KUKA KRL program: EPS_2_251349_CBMH080_A_20251001124254.src

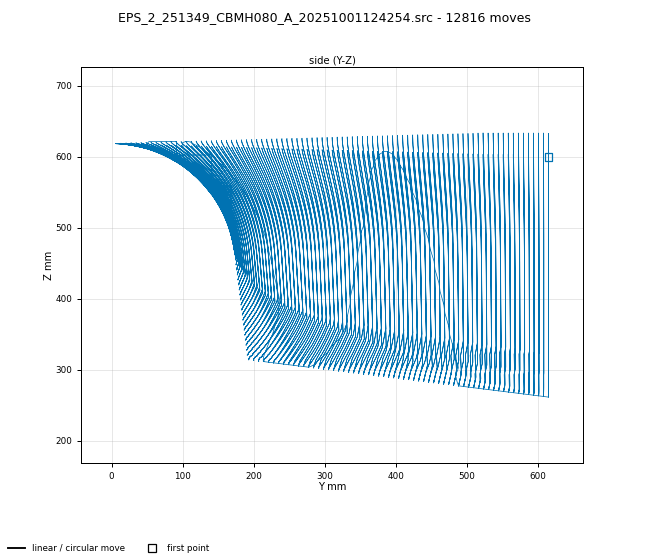
[picture p0: tool path of EPS_2_251349_CBMH080_A_20251001124254.src, 12816 of 12818 moves have a stored position in this frame; points joined in program order, loops and branches not executed]
&ACCESS RVP
&REL 4
&COMMENT QRS 19112012
&PARAM EDITMASK = *
DEF PART()
EXT BAS (BAS_COMMAND :IN,REAL :IN )
INT I
BAS (#INITMOV,0 )

;KUKA QRS Post kuka4.cps  Date:22-06-2017 !

File_ID=2857

QRS_PRE_INIT()

;Init var - Until changes are made in qrs_pre_init
Outlet_Square_prg=0
Inlet_1_Square_prg=0
Inlet_2_Square_prg=0
Inlet_3_Square_prg=0
Inlet_4_Square_prg=0
Inlet_5_Square_prg=0

Outlet_1={X 0.000, Y 523.550, Z 484.000, B 0.000, E1 0.000 }
Inlet_1={X 0.000, Y 525.740, Z 454.000, B 0.000, E1 180.000 }
Outlet_1_type=299
Inlet_1_type=299
;QRS#1=Sidecore dimensions
;QRS#2=300-12" PVC SDR 35
;QRS#3=300-12" PVC SDR 35
;QRS#4=
;QRS#5=
;QRS#6=
;QRS#7=
;QRS#8=
;QRS#9=16M PSX
;QRS#10=16M PSX
;QRS#11=
;QRS#12=
;QRS#13=
;QRS#14=
;QRS#15=
;QRS#16=1220x127x914 3'
;QRS#17=EPS Height
;QRS#18=633,5
;QRS#19=*
;QRS#20= UPDATED VERSION 22-06-2017
;QRS#21=*
Outlet_Square=0150
Inlet_1_Square=0150
Inlet_2_Square=0
Inlet_3_Square=0
Inlet_4_Square=0
Inlet_5_Square=0
Mill_Square=1
Outlet_Square_Prg=206
Inlet_1_Square_prg=206

QRS_INIT()

$ADVANCE=5

; T1
PTP {E1 173.644,E2 173.644}
PTP {X 0,Y 615.424,A -85,B 0,C 180,E1 173.644,E2 173.644,E3 0,E4 0,E5 0,E6 0}
QRS_SPEED_INIT()
LIN {X 0,Y 615.424,Z 600,A -85,B 0,C 180,E1 173.644,E2 173.644,E3 0,E4 0,E5 0,E6 0} C_VEL
LIN {X 0,Y 615.424,Z 271.5,A -85,B 0,C 180,E1 173.644,E2 173.644} C_VEL
LIN {X 0,Y 615.424,Z 263.323,A -85,B 0,C 180,E1 173.644,E2 173.644} C_VEL
LIN {X 0,Y 615.426,Z 261.323,A -85,B 0,C 180,E1 173.458,E2 173.458} C_VEL
LIN {X 0,Y 615.491,Z 261.325,A -85,B 0,C 180,E1 170.801,E2 170.801} C_VEL
LIN {X 0,Y 615.447,Z 261.319,A -85,B 0,C 180,E1 168.138,E2 168.138} C_VEL
LIN {X 0,Y 615.442,Z 261.319,A -85,B 0,C 180,E1 166.078,E2 166.078} C_VEL
LIN {X 0,Y 615.442,Z 261.319,A -85,B 0,C 180,E1 164.094,E2 164.094} C_VEL
LIN {X 0,Y 615.44,Z 261.319,A -85,B 0,C 180,E1 162.042,E2 162.042} C_VEL
LIN {X 0,Y 615.435,Z 261.319,A -85,B 0,C 180,E1 159.965,E2 159.965} C_VEL
LIN {X 0,Y 615.434,Z 261.321,A -85,B 0,C 180,E1 157.662,E2 157.662} C_VEL
LIN {X 0,Y 615.491,Z 261.325,A -85,B 0,C 180,E1 155.008,E2 155.008} C_VEL
LIN {X 0,Y 615.494,Z 261.32,A -85,B 0,C 180,E1 152.823,E2 152.823} C_VEL
LIN {X 0,Y 615.451,Z 261.316,A -85,B 0,C 180,E1 150.209,E2 150.209} C_VEL
LIN {X 0,Y 615.44,Z 261.321,A -85,B 0,C 180,E1 147.674,E2 147.674} C_VEL
LIN {X 0,Y 615.485,Z 261.325,A -85,B 0,C 180,E1 145.185,E2 145.185} C_VEL
LIN {X 0,Y 615.491,Z 261.315,A -85,B 0,C 180,E1 142.758,E2 142.758} C_VEL
LIN {X 0,Y 615.453,Z 261.315,A -85,B 0,C 180,E1 140.247,E2 140.247} C_VEL
LIN {X 0,Y 615.455,Z 261.321,A -85,B 0,C 180,E1 137.644,E2 137.644} C_VEL
LIN {X 0,Y 615.489,Z 261.317,A -85,B 0,C 180,E1 134.931,E2 134.931} C_VEL
LIN {X 0,Y 615.455,Z 261.315,A -85,B 0,C 180,E1 132.354,E2 132.354} C_VEL
LIN {X 0,Y 615.457,Z 261.32,A -85,B 0,C 180,E1 129.751,E2 129.751} C_VEL
LIN {X 0,Y 615.488,Z 261.315,A -85,B 0,C 180,E1 126.937,E2 126.937} C_VEL
LIN {X 0,Y 615.453,Z 261.318,A -85,B 0,C 180,E1 124.023,E2 124.023} C_VEL
LIN {X 0,Y 615.492,Z 261.316,A -85,B 0,C 180,E1 121.086,E2 121.086} C_VEL
LIN {X 0,Y 615.462,Z 261.313,A -85,B 0,C 180,E1 118.446,E2 118.446} C_VEL
LIN {X 0,Y 615.476,Z 261.322,A -85,B 0,C 180,E1 115.715,E2 115.715} C_VEL
LIN {X 0,Y 615.486,Z 261.31,A -85,B 0,C 180,E1 112.844,E2 112.844} C_VEL
LIN {X 0,Y 615.459,Z 261.362,A -85,B 0,C 180,E1 112.263,E2 112.263} C_VEL
LIN {X 0,Y 615.464,Z 281.213,A -85,B 0,C 180,E1 109.685,E2 109.685} C_VEL
LIN {X 0,Y 615.457,Z 292.799,A -85,B 0,C 180,E1 108.199,E2 108.199} C_VEL
LIN {X 0,Y 615.489,Z 457.351,A -85,B 0,C 180,E1 106.199,E2 106.199} C_VEL
LIN {X 0,Y 615.489,Z 471.838,A -85,B 0,C 180,E1 105.905,E2 105.905} C_VEL
LIN {X 0,Y 615.477,Z 486.432,A -85,B 0,C 180,E1 105.48,E2 105.48} C_VEL
LIN {X 0,Y 615.491,Z 499.749,A -85,B 0,C 180,E1 104.971,E2 104.971} C_VEL
LIN {X 0,Y 615.483,Z 513.386,A -85,B 0,C 180,E1 104.319,E2 104.319} C_VEL
LIN {X 0,Y 615.5,Z 526.673,A -85,B 0,C 180,E1 103.537,E2 103.537} C_VEL
LIN {X 0,Y 615.497,Z 538.522,A -85,B 0,C 180,E1 102.697,E2 102.697} C_VEL
LIN {X 0,Y 615.497,Z 550.364,A -85,B 0,C 180,E1 101.693,E2 101.693} C_VEL
LIN {X 0,Y 615.495,Z 560.168,A -85,B 0,C 180,E1 100.708,E2 100.708} C_VEL
LIN {X 0,Y 615.495,Z 570.015,A -85,B 0,C 180,E1 99.53,E2 99.53} C_VEL
LIN {X 0,Y 615.497,Z 578.104,A -85,B 0,C 180,E1 98.371,E2 98.371} C_VEL
LIN {X 0,Y 615.491,Z 584.784,A -85,B 0,C 180,E1 97.215,E2 97.215} C_VEL
LIN {X 0,Y 615.497,Z 590.949,A -85,B 0,C 180,E1 95.898,E2 95.898} C_VEL
LIN {X 0,Y 615.49,Z 595.717,A -85,B 0,C 180,E1 94.584,E2 94.584} C_VEL
LIN {X 0,Y 615.491,Z 599.221,A -85,B 0,C 180,E1 93.273,E2 93.273} C_VEL
LIN {X 0,Y 615.499,Z 601.54,A -85,B 0,C 180,E1 91.963,E2 91.963} C_VEL
LIN {X 0,Y 615.491,Z 602.728,A -85,B 0,C 180,E1 90.654,E2 90.654} C_VEL
LIN {X 0,Y 615.492,Z 602.751,A -85,B 0,C 180,E1 89.346,E2 89.346} C_VEL
LIN {X 0,Y 615.499,Z 601.646,A -85,B 0,C 180,E1 88.037,E2 88.037} C_VEL
LIN {X 0,Y 615.494,Z 599.416,A -85,B 0,C 180,E1 86.727,E2 86.727} C_VEL
LIN {X 0,Y 615.491,Z 596.005,A -85,B 0,C 180,E1 85.416,E2 85.416} C_VEL
LIN {X 0,Y 615.498,Z 591.336,A -85,B 0,C 180,E1 84.102,E2 84.102} C_VEL
LIN {X 0,Y 615.49,Z 585.273,A -85,B 0,C 180,E1 82.785,E2 82.785} C_VEL
LIN {X 0,Y 615.49,Z 577.635,A -85,B 0,C 180,E1 81.464,E2 81.464} C_VEL
LIN {X 0,Y 615.495,Z 569.452,A -85,B 0,C 180,E1 80.304,E2 80.304} C_VEL
LIN {X 0,Y 615.496,Z 559.333,A -85,B 0,C 180,E1 79.109,E2 79.109} C_VEL
LIN {X 0,Y 615.498,Z 547.686,A -85,B 0,C 180,E1 77.973,E2 77.973} C_VEL
LIN {X 0,Y 615.498,Z 536.417,A -85,B 0,C 180,E1 77.051,E2 77.051} C_VEL
LIN {X 0,Y 615.498,Z 524.179,A -85,B 0,C 180,E1 76.211,E2 76.211} C_VEL
LIN {X 0,Y 615.48,Z 510.782,A -85,B 0,C 180,E1 75.451,E2 75.451} C_VEL
LIN {X 0,Y 615.493,Z 496.919,A -85,B 0,C 180,E1 74.817,E2 74.817} C_VEL
LIN {X 0,Y 615.488,Z 482.706,A -85,B 0,C 180,E1 74.308,E2 74.308} C_VEL
LIN {X 0,Y 615.497,Z 468.664,A -85,B 0,C 180,E1 73.932,E2 73.932} C_VEL
LIN {X 0,Y 615.487,Z 453.239,A -85,B 0,C 180,E1 73.653,E2 73.653} C_VEL
LIN {X 0,Y 615.457,Z 292.88,A -85,B 0,C 180,E1 71.721,E2 71.721} C_VEL
LIN {X 0,Y 615.49,Z 271.117,A -85,B 0,C 180,E1 68.92,E2 68.92} C_VEL
LIN {X 0,Y 615.465,Z 261.314,A -85,B 0,C 180,E1 67.628,E2 67.628} C_VEL
LIN {X 0,Y 615.491,Z 261.31,A -85,B 0,C 180,E1 65.009,E2 65.009} C_VEL
LIN {X 0,Y 615.467,Z 261.32,A -85,B 0,C 180,E1 62.085,E2 62.085} C_VEL
LIN {X 0,Y 615.458,Z 261.316,A -85,B 0,C 180,E1 59.839,E2 59.839} C_VEL
LIN {X 0,Y 615.468,Z 261.312,A -85,B 0,C 180,E1 57.542,E2 57.542} C_VEL
LIN {X 0,Y 615.499,Z 261.308,A -85,B 0,C 180,E1 55.187,E2 55.187} C_VEL
LIN {X 0,Y 615.493,Z 261.321,A -85,B 0,C 180,E1 52.759,E2 52.759} C_VEL
LIN {X 0,Y 615.465,Z 261.321,A -85,B 0,C 180,E1 50.249,E2 50.249} C_VEL
LIN {X 0,Y 615.458,Z 261.314,A -85,B 0,C 180,E1 47.646,E2 47.646} C_VEL
LIN {X 0,Y 615.489,Z 261.319,A -85,B 0,C 180,E1 44.933,E2 44.933} C_VEL
LIN {X 0,Y 615.462,Z 261.321,A -85,B 0,C 180,E1 42.355,E2 42.355} C_VEL
LIN {X 0,Y 615.456,Z 261.315,A -85,B 0,C 180,E1 39.753,E2 39.753} C_VEL
LIN {X 0,Y 615.489,Z 261.323,A -85,B 0,C 180,E1 36.939,E2 36.939} C_VEL
LIN {X 0,Y 615.446,Z 261.317,A -85,B 0,C 180,E1 34.025,E2 34.025} C_VEL
LIN {X 0,Y 615.492,Z 261.32,A -85,B 0,C 180,E1 31.089,E2 31.089} C_VEL
LIN {X 0,Y 615.451,Z 261.321,A -85,B 0,C 180,E1 28.447,E2 28.447} C_VEL
LIN {X 0,Y 615.449,Z 261.321,A -85,B 0,C 180,E1 26.446,E2 26.446} C_VEL
LIN {X 0,Y 615.442,Z 261.318,A -85,B 0,C 180,E1 24.002,E2 24.002} C_VEL
LIN {X 0,Y 615.491,Z 261.314,A -85,B 0,C 180,E1 21.432,E2 21.432} C_VEL
LIN {X 0,Y 615.448,Z 261.322,A -85,B 0,C 180,E1 18.599,E2 18.599} C_VEL
LIN {X 0,Y 615.436,Z 261.321,A -85,B 0,C 180,E1 16.42,E2 16.42} C_VEL
LIN {X 0,Y 615.44,Z 261.322,A -85,B 0,C 180,E1 14.55,E2 14.55} C_VEL
LIN {X 0,Y 615.437,Z 261.322,A -85,B 0,C 180,E1 12.531,E2 12.531} C_VEL
LIN {X 0,Y 615.434,Z 261.322,A -85,B 0,C 180,E1 10.528,E2 10.528} C_VEL
LIN {X 0,Y 615.429,Z 261.323,A -85,B 0,C 180,E1 8.538,E2 8.538} C_VEL
LIN {X 0,Y 615.431,Z 261.322,A -85,B 0,C 180,E1 6.546,E2 6.546} C_VEL
LIN {X 0,Y 615.427,Z 261.323,A -85,B 0,C 180,E1 4.585,E2 4.585} C_VEL
LIN {X 0,Y 615.43,Z 261.323,A -85,B 0,C 180,E1 2.618,E2 2.618} C_VEL
LIN {X 0,Y 615.429,Z 261.323,A -85,B 0,C 180,E1 0.654,E2 0.654} C_VEL
LIN {X 0,Y 615.428,Z 261.323,A -85,B 0,C 180,E1 -1.309,E2 -1.309} C_VEL
LIN {X 0,Y 615.428,Z 261.323,A -85,B 0,C 180,E1 -3.273,E2 -3.273} C_VEL
LIN {X 0,Y 615.426,Z 261.324,A -85,B 0,C 180,E1 -5.242,E2 -5.242} C_VEL
LIN {X 0,Y 615.426,Z 261.324,A -85,B 0,C 180,E1 -7.216,E2 -7.216} C_VEL
LIN {X 0,Y 615.423,Z 261.324,A -85,B 0,C 180,E1 -9.2,E2 -9.2} C_VEL
LIN {X 0,Y 615.422,Z 261.324,A -85,B 0,C 180,E1 -11.194,E2 -11.194} C_VEL
LIN {X 0,Y 615.419,Z 261.324,A -85,B 0,C 180,E1 -13.203,E2 -13.203} C_VEL
LIN {X 0,Y 615.416,Z 261.325,A -85,B 0,C 180,E1 -15.228,E2 -15.228} C_VEL
LIN {X 0,Y 615.412,Z 261.325,A -85,B 0,C 180,E1 -17.273,E2 -17.273} C_VEL
LIN {X 0,Y 615.41,Z 261.325,A -85,B 0,C 180,E1 -19.34,E2 -19.34} C_VEL
LIN {X 0,Y 615.411,Z 261.325,A -85,B 0,C 180,E1 -21.435,E2 -21.435} C_VEL
LIN {X 0,Y 615.416,Z 261.325,A -85,B 0,C 180,E1 -23.559,E2 -23.559} C_VEL
LIN {X 0,Y 615.485,Z 261.323,A -85,B 0,C 180,E1 -26.444,E2 -26.444} C_VEL
LIN {X 0,Y 615.454,Z 261.322,A -85,B 0,C 180,E1 -28.66,E2 -28.66} C_VEL
LIN {X 0,Y 615.422,Z 261.323,A -85,B 0,C 180,E1 -31.078,E2 -31.078} C_VEL
LIN {X 0,Y 615.42,Z 261.323,A -85,B 0,C 180,E1 -33.24,E2 -33.24} C_VEL
LIN {X 0,Y 615.454,Z 261.324,A -85,B 0,C 180,E1 -35.832,E2 -35.832} C_VEL
LIN {X 0,Y 615.486,Z 261.326,A -85,B 0,C 180,E1 -38.069,E2 -38.069} C_VEL
LIN {X 0,Y 615.455,Z 261.32,A -85,B 0,C 180,E1 -40.609,E2 -40.609} C_VEL
LIN {X 0,Y 615.428,Z 261.321,A -85,B 0,C 180,E1 -43.043,E2 -43.043} C_VEL
LIN {X 0,Y 615.428,Z 261.321,A -85,B 0,C 180,E1 -45.074,E2 -45.074} C_VEL
LIN {X 0,Y 615.455,Z 261.323,A -85,B 0,C 180,E1 -47.646,E2 -47.646} C_VEL
LIN {X 0,Y 615.492,Z 261.317,A -85,B 0,C 180,E1 -50.252,E2 -50.252} C_VEL
LIN {X 0,Y 615.441,Z 261.318,A -85,B 0,C 180,E1 -52.756,E2 -52.756} C_VEL
LIN {X 0,Y 615.437,Z 261.321,A -85,B 0,C 180,E1 -55.183,E2 -55.183} C_VEL
LIN {X 0,Y 615.476,Z 261.324,A -85,B 0,C 180,E1 -57.671,E2 -57.671} C_VEL
LIN {X 0,Y 615.453,Z 261.316,A -85,B 0,C 180,E1 -60.593,E2 -60.593} C_VEL
LIN {X 0,Y 615.44,Z 261.319,A -85,B 0,C 180,E1 -62.964,E2 -62.964} C_VEL
LIN {X 0,Y 615.441,Z 261.446,A -85,B 0,C 180,E1 -64.936,E2 -64.936} C_VEL
LIN {X 0,Y 615.482,Z 284.083,A -85,B 0,C 180,E1 -67.53,E2 -67.53} C_VEL
LIN {X 0,Y 615.49,Z 308.881,A -85,B 0,C 180,E1 -70.316,E2 -70.316} C_VEL
LIN {X 0,Y 615.488,Z 322.06,A -85,B 0,C 180,E1 -71.762,E2 -71.762} C_VEL
LIN {X 0,Y 615.487,Z 488.129,A -85,B 0,C 180,E1 -73.767,E2 -73.767} C_VEL
LIN {X 0,Y 615.49,Z 503.731,A -85,B 0,C 180,E1 -74.095,E2 -74.095} C_VEL
LIN {X 0,Y 615.48,Z 519.063,A -85,B 0,C 180,E1 -74.562,E2 -74.562} C_VEL
LIN {X 0,Y 615.492,Z 532.764,A -85,B 0,C 180,E1 -75.113,E2 -75.113} C_VEL
LIN {X 0,Y 615.494,Z 547.049,A -85,B 0,C 180,E1 -75.834,E2 -75.834} C_VEL
LIN {X 0,Y 615.497,Z 559.904,A -85,B 0,C 180,E1 -76.631,E2 -76.631} C_VEL
LIN {X 0,Y 615.495,Z 572.259,A -85,B 0,C 180,E1 -77.554,E2 -77.554} C_VEL
LIN {X 0,Y 615.495,Z 582.61,A -85,B 0,C 180,E1 -78.474,E2 -78.474} C_VEL
LIN {X 0,Y 615.495,Z 592.187,A -85,B 0,C 180,E1 -79.474,E2 -79.474} C_VEL
LIN {X 0,Y 615.494,Z 601.579,A -85,B 0,C 180,E1 -80.636,E2 -80.636} C_VEL
LIN {X 0,Y 615.495,Z 609.382,A -85,B 0,C 180,E1 -81.794,E2 -81.794} C_VEL
LIN {X 0,Y 615.496,Z 616.607,A -85,B 0,C 180,E1 -83.102,E2 -83.102} C_VEL
LIN {X 0,Y 615.499,Z 622.437,A -85,B 0,C 180,E1 -84.43,E2 -84.43} C_VEL
LIN {X 0,Y 615.491,Z 625.861,A -85,B 0,C 180,E1 -85.416,E2 -85.416} C_VEL
LIN {X 0,Y 615.492,Z 629.318,A -85,B 0,C 180,E1 -86.727,E2 -86.727} C_VEL
LIN {X 0,Y 615.497,Z 631.593,A -85,B 0,C 180,E1 -88.037,E2 -88.037} C_VEL
LIN {X 0,Y 615.493,Z 632.74,A -85,B 0,C 180,E1 -89.346,E2 -89.346} C_VEL
LIN {X 0,Y 615.493,Z 632.74,A -85,B 0,C 180,E1 -90.654,E2 -90.654} C_VEL
LIN {X 0,Y 615.497,Z 631.593,A -85,B 0,C 180,E1 -91.963,E2 -91.963} C_VEL
LIN {X 0,Y 615.492,Z 629.318,A -85,B 0,C 180,E1 -93.273,E2 -93.273} C_VEL
LIN {X 0,Y 615.491,Z 625.861,A -85,B 0,C 180,E1 -94.584,E2 -94.584} C_VEL
LIN {X 0,Y 615.49,Z 621.144,A -85,B 0,C 180,E1 -95.898,E2 -95.898} C_VEL
LIN {X 0,Y 615.495,Z 615.03,A -85,B 0,C 180,E1 -97.215,E2 -97.215} C_VEL
LIN {X 0,Y 615.49,Z 607.335,A -85,B 0,C 180,E1 -98.536,E2 -98.536} C_VEL
LIN {X 0,Y 615.495,Z 599.116,A -85,B 0,C 180,E1 -99.696,E2 -99.696} C_VEL
LIN {X 0,Y 615.497,Z 588.895,A -85,B 0,C 180,E1 -100.893,E2 -100.893} C_VEL
LIN {X 0,Y 615.495,Z 579.071,A -85,B 0,C 180,E1 -101.86,E2 -101.86} C_VEL
LIN {X 0,Y 615.498,Z 566.952,A -85,B 0,C 180,E1 -102.865,E2 -102.865} C_VEL
LIN {X 0,Y 615.498,Z 554.804,A -85,B 0,C 180,E1 -103.705,E2 -103.705} C_VEL
LIN {X 0,Y 615.484,Z 541.386,A -85,B 0,C 180,E1 -104.472,E2 -104.472} C_VEL
LIN {X 0,Y 615.495,Z 526.858,A -85,B 0,C 180,E1 -105.141,E2 -105.141} C_VEL
LIN {X 0,Y 615.484,Z 512.629,A -85,B 0,C 180,E1 -105.65,E2 -105.65} C_VEL
LIN {X 0,Y 615.499,Z 498.141,A -85,B 0,C 180,E1 -106.035,E2 -106.035} C_VEL
LIN {X 0,Y 615.487,Z 483.539,A -85,B 0,C 180,E1 -106.298,E2 -106.298} C_VEL
LIN {X 0,Y 615.489,Z 321.746,A -85,B 0,C 180,E1 -108.258,E2 -108.258} C_VEL
LIN {X 0,Y 615.49,Z 296.397,A -85,B 0,C 180,E1 -111.08,E2 -111.08} C_VEL
LIN {X 0,Y 615.495,Z 270.579,A -85,B 0,C 180,E1 -114.01,E2 -114.01} C_VEL
LIN {X 0,Y 615.441,Z 261.318,A -85,B 0,C 180,E1 -115.1,E2 -115.1} C_VEL
LIN {X 0,Y 615.489,Z 261.317,A -85,B 0,C 180,E1 -117.914,E2 -117.914} C_VEL
LIN {X 0,Y 615.499,Z 261.324,A -85,B 0,C 180,E1 -120.159,E2 -120.159} C_VEL
LIN {X 0,Y 615.462,Z 261.323,A -85,B 0,C 180,E1 -122.458,E2 -122.458} C_VEL
LIN {X 0,Y 615.437,Z 261.321,A -85,B 0,C 180,E1 -124.817,E2 -124.817} C_VEL
LIN {X 0,Y 615.442,Z 261.318,A -85,B 0,C 180,E1 -127.244,E2 -127.244} C_VEL
LIN {X 0,Y 615.495,Z 261.325,A -85,B 0,C 180,E1 -130.09,E2 -130.09} C_VEL
LIN {X 0,Y 615.457,Z 261.323,A -85,B 0,C 180,E1 -132.354,E2 -132.354} C_VEL
LIN {X 0,Y 615.429,Z 261.321,A -85,B 0,C 180,E1 -134.926,E2 -134.926} C_VEL
LIN {X 0,Y 615.429,Z 261.321,A -85,B 0,C 180,E1 -136.957,E2 -136.957} C_VEL
LIN {X 0,Y 615.456,Z 261.319,A -85,B 0,C 180,E1 -139.391,E2 -139.391} C_VEL
LIN {X 0,Y 615.478,Z 261.326,A -85,B 0,C 180,E1 -141.987,E2 -141.987} C_VEL
LIN {X 0,Y 615.434,Z 261.324,A -85,B 0,C 180,E1 -144.381,E2 -144.381} C_VEL
LIN {X 0,Y 615.421,Z 261.322,A -85,B 0,C 180,E1 -146.76,E2 -146.76} C_VEL
LIN {X 0,Y 615.431,Z 261.322,A -85,B 0,C 180,E1 -149.077,E2 -149.077} C_VEL
LIN {X 0,Y 615.483,Z 261.321,A -85,B 0,C 180,E1 -151.548,E2 -151.548} C_VEL
LIN {X 0,Y 615.431,Z 261.324,A -85,B 0,C 180,E1 -154.282,E2 -154.282} C_VEL
LIN {X 0,Y 615.419,Z 261.324,A -85,B 0,C 180,E1 -156.441,E2 -156.441} C_VEL
LIN {X 0,Y 615.414,Z 261.324,A -85,B 0,C 180,E1 -158.565,E2 -158.565} C_VEL
LIN {X 0,Y 615.412,Z 261.324,A -85,B 0,C 180,E1 -160.66,E2 -160.66} C_VEL
LIN {X 0,Y 615.481,Z 261.328,A -85,B 0,C 180,E1 -163.566,E2 -163.566} C_VEL
LIN {X 0,Y 615.428,Z 261.325,A -85,B 0,C 180,E1 -166.125,E2 -166.125} C_VEL
LIN {X 0,Y 615.426,Z 261.325,A -85,B 0,C 180,E1 -168.138,E2 -168.138} C_VEL
LIN {X 0,Y 615.425,Z 261.324,A -85,B 0,C 180,E1 -170.137,E2 -170.137} C_VEL
LIN {X 0,Y 615.428,Z 261.324,A -85,B 0,C 180,E1 -172.124,E2 -172.124} C_VEL
LIN {X 0,Y 615.43,Z 261.323,A -85,B 0,C 180,E1 -174.101,E2 -174.101} C_VEL
LIN {X 0,Y 615.431,Z 261.323,A -85,B 0,C 180,E1 -176.071,E2 -176.071} C_VEL
LIN {X 0,Y 615.434,Z 261.322,A -85,B 0,C 180,E1 -178.037,E2 -178.037} C_VEL
LIN {X 0,Y 615.437,Z 261.322,A -85,B 0,C 180,E1 -180,E2 -180} C_VEL
LIN {X 0,Y 615.44,Z 261.321,A -85,B 0,C 180,E1 -181.963,E2 -181.963} C_VEL
LIN {X 0,Y 615.441,Z 261.321,A -85,B 0,C 180,E1 -183.929,E2 -183.929} C_VEL
LIN {X 0,Y 615.445,Z 261.32,A -85,B 0,C 180,E1 -185.899,E2 -185.899} C_VEL
LIN {X 0,Y 615.426,Z 261.323,A -85,B 0,C 180,E1 -186.542,E2 -186.542} C_VEL
LIN {X 0,Y 614.793,Z 261.474,A -85,B 0,C 180,E1 -187.088,E2 -187.088} C_VEL
LIN {X 0,Y 611.998,Z 261.872,A -85,B 0,C 180,E1 -187.975,E2 -187.975} C_VEL
LIN {X 0,Y 609.606,Z 262.189,A -85,B 0,C 180,E1 -188.687,E2 -188.687} C_VEL
LIN {X 0,Y 608.551,Z 262.311,A -85,B 0,C 180,E1 -189.237,E2 -189.237} C_VEL
LIN {X 0,Y 608.452,Z 262.32,A -85,B 0,C 180,E1 -189.423,E2 -189.423} C_VEL
LIN {X 0,Y 608.422,Z 262.317,A -85,B 0,C 180,E1 -192.001,E2 -192.001} C_VEL
LIN {X 0,Y 608.406,Z 262.318,A -85,B 0,C 180,E1 -194.039,E2 -194.039} C_VEL
LIN {X 0,Y 608.43,Z 262.317,A -85,B 0,C 180,E1 -196.522,E2 -196.522} C_VEL
LIN {X 0,Y 608.436,Z 262.317,A -85,B 0,C 180,E1 -199.571,E2 -199.571} C_VEL
LIN {X 0,Y 608.419,Z 262.318,A -85,B 0,C 180,E1 -202.408,E2 -202.408} C_VEL
LIN {X 0,Y 608.444,Z 262.319,A -85,B 0,C 180,E1 -205.301,E2 -205.301} C_VEL
LIN {X 0,Y 608.434,Z 262.317,A -85,B 0,C 180,E1 -207.519,E2 -207.519} C_VEL
LIN {X 0,Y 608.414,Z 262.317,A -85,B 0,C 180,E1 -209.965,E2 -209.965} C_VEL
LIN {X 0,Y 608.427,Z 262.319,A -85,B 0,C 180,E1 -212.52,E2 -212.52} C_VEL
LIN {X 0,Y 608.43,Z 262.32,A -85,B 0,C 180,E1 -215.279,E2 -215.279} C_VEL
LIN {X 0,Y 608.444,Z 262.313,A -85,B 0,C 180,E1 -217.748,E2 -217.748} C_VEL
LIN {X 0,Y 608.423,Z 262.319,A -85,B 0,C 180,E1 -220.328,E2 -220.328} C_VEL
LIN {X 0,Y 608.456,Z 262.32,A -85,B 0,C 180,E1 -222.96,E2 -222.96} C_VEL
LIN {X 0,Y 608.425,Z 262.316,A -85,B 0,C 180,E1 -225.739,E2 -225.739} C_VEL
LIN {X 0,Y 608.428,Z 262.316,A -85,B 0,C 180,E1 -227.937,E2 -227.937} C_VEL
LIN {X 0,Y 608.443,Z 262.324,A -85,B 0,C 180,E1 -230.706,E2 -230.706} C_VEL
LIN {X 0,Y 608.458,Z 262.315,A -85,B 0,C 180,E1 -233.086,E2 -233.086} C_VEL
LIN {X 0,Y 608.461,Z 262.311,A -85,B 0,C 180,E1 -235.531,E2 -235.531} C_VEL
LIN {X 0,Y 608.445,Z 262.314,A -85,B 0,C 180,E1 -237.905,E2 -237.905} C_VEL
LIN {X 0,Y 608.45,Z 262.317,A -85,B 0,C 180,E1 -240.22,E2 -240.22} C_VEL
LIN {X 0,Y 608.484,Z 262.315,A -85,B 0,C 180,E1 -242.792,E2 -242.792} C_VEL
LIN {X 0,Y 608.442,Z 262.314,A -85,B 0,C 180,E1 -245.429,E2 -245.429} C_VEL
LIN {X 0,Y 608.436,Z 262.334,A -85,B 0,C 180,E1 -247.594,E2 -247.594} C_VEL
LIN {X 0,Y 608.577,Z 277.311,A -85,B 0,C 180,E1 -249.572,E2 -249.572} C_VEL
LIN {X 0,Y 608.516,Z 292.824,A -85,B 0,C 180,E1 -251.586,E2 -251.586} C_VEL
LIN {X 0,Y 608.715,Z 296.703,A -85,B 0,C 180,E1 -251.654,E2 -251.654} C_VEL
LIN {X 0,Y 608.684,Z 458.428,A -85,B 0,C 180,E1 -253.631,E2 -253.631} C_VEL
LIN {X 0,Y 608.647,Z 473.657,A -85,B 0,C 180,E1 -253.955,E2 -253.955} C_VEL
LIN {X 0,Y 608.61,Z 489.006,A -85,B 0,C 180,E1 -254.426,E2 -254.426} C_VEL
LIN {X 0,Y 608.589,Z 503.684,A -85,B 0,C 180,E1 -255.026,E2 -255.026} C_VEL
LIN {X 0,Y 608.57,Z 517.448,A -85,B 0,C 180,E1 -255.735,E2 -255.735} C_VEL
LIN {X 0,Y 608.547,Z 530.55,A -85,B 0,C 180,E1 -256.561,E2 -256.561} C_VEL
LIN {X 0,Y 608.505,Z 542.845,A -85,B 0,C 180,E1 -257.494,E2 -257.494} C_VEL
LIN {X 0,Y 608.497,Z 554.054,A -85,B 0,C 180,E1 -258.508,E2 -258.508} C_VEL
LIN {X 0,Y 608.477,Z 564.937,A -85,B 0,C 180,E1 -259.687,E2 -259.687} C_VEL
LIN {X 0,Y 608.469,Z 573.986,A -85,B 0,C 180,E1 -260.862,E2 -260.862} C_VEL
LIN {X 0,Y 608.459,Z 581.481,A -85,B 0,C 180,E1 -262.033,E2 -262.033} C_VEL
LIN {X 0,Y 608.445,Z 588.63,A -85,B 0,C 180,E1 -263.397,E2 -263.397} C_VEL
LIN {X 0,Y 608.436,Z 593.994,A -85,B 0,C 180,E1 -264.698,E2 -264.698} C_VEL
LIN {X 0,Y 608.432,Z 598.168,A -85,B 0,C 180,E1 -266.026,E2 -266.026} C_VEL
LIN {X 0,Y 608.421,Z 601.11,A -85,B 0,C 180,E1 -267.352,E2 -267.352} C_VEL
LIN {X 0,Y 608.444,Z 602.88,A -85,B 0,C 180,E1 -268.676,E2 -268.676} C_VEL
LIN {X 0,Y 608.432,Z 603.495,A -85,B 0,C 180,E1 -270,E2 -270} C_VEL
LIN {X 0,Y 608.446,Z 602.944,A -85,B 0,C 180,E1 -271.324,E2 -271.324} C_VEL
LIN {X 0,Y 608.424,Z 601.259,A -85,B 0,C 180,E1 -272.648,E2 -272.648} C_VEL
LIN {X 0,Y 608.432,Z 598.408,A -85,B 0,C 180,E1 -273.974,E2 -273.974} C_VEL
LIN {X 0,Y 608.436,Z 594.329,A -85,B 0,C 180,E1 -275.302,E2 -275.302} C_VEL
LIN {X 0,Y 608.445,Z 588.922,A -85,B 0,C 180,E1 -276.633,E2 -276.633} C_VEL
LIN {X 0,Y 608.457,Z 582.024,A -85,B 0,C 180,E1 -277.967,E2 -277.967} C_VEL
LIN {X 0,Y 608.466,Z 574.593,A -85,B 0,C 180,E1 -279.138,E2 -279.138} C_VEL
LIN {X 0,Y 608.476,Z 565.665,A -85,B 0,C 180,E1 -280.313,E2 -280.313} C_VEL
LIN {X 0,Y 608.496,Z 554.95,A -85,B 0,C 180,E1 -281.492,E2 -281.492} C_VEL
LIN {X 0,Y 608.513,Z 542.91,A -85,B 0,C 180,E1 -282.591,E2 -282.591} C_VEL
LIN {X 0,Y 608.543,Z 530.623,A -85,B 0,C 180,E1 -283.524,E2 -283.524} C_VEL
LIN {X 0,Y 608.584,Z 517.682,A -85,B 0,C 180,E1 -284.341,E2 -284.341} C_VEL
LIN {X 0,Y 608.606,Z 503.778,A -85,B 0,C 180,E1 -285.059,E2 -285.059} C_VEL
LIN {X 0,Y 608.638,Z 489.118,A -85,B 0,C 180,E1 -285.659,E2 -285.659} C_VEL
LIN {X 0,Y 608.666,Z 473.547,A -85,B 0,C 180,E1 -286.138,E2 -286.138} C_VEL
LIN {X 0,Y 608.687,Z 457.547,A -85,B 0,C 180,E1 -286.473,E2 -286.473} C_VEL
LIN {X 0,Y 608.717,Z 294.118,A -85,B 0,C 180,E1 -288.468,E2 -288.468} C_VEL
LIN {X 0,Y 608.512,Z 292.897,A -85,B 0,C 180,E1 -288.495,E2 -288.495} C_VEL
LIN {X 0,Y 608.565,Z 272.464,A -85,B 0,C 180,E1 -291.154,E2 -291.154} C_VEL
LIN {X 0,Y 608.451,Z 262.315,A -85,B 0,C 180,E1 -292.501,E2 -292.501} C_VEL
LIN {X 0,Y 608.459,Z 262.318,A -85,B 0,C 180,E1 -295.3,E2 -295.3} C_VEL
LIN {X 0,Y 608.443,Z 262.324,A -85,B 0,C 180,E1 -297.517,E2 -297.517} C_VEL
LIN {X 0,Y 608.434,Z 262.318,A -85,B 0,C 180,E1 -299.966,E2 -299.966} C_VEL
LIN {X 0,Y 608.446,Z 262.313,A -85,B 0,C 180,E1 -302.52,E2 -302.52} C_VEL
LIN {X 0,Y 608.446,Z 262.321,A -85,B 0,C 180,E1 -305.276,E2 -305.276} C_VEL
LIN {X 0,Y 608.453,Z 262.317,A -85,B 0,C 180,E1 -307.746,E2 -307.746} C_VEL
LIN {X 0,Y 608.43,Z 262.315,A -85,B 0,C 180,E1 -310.326,E2 -310.326} C_VEL
LIN {X 0,Y 608.453,Z 262.317,A -85,B 0,C 180,E1 -312.958,E2 -312.958} C_VEL
LIN {X 0,Y 608.428,Z 262.319,A -85,B 0,C 180,E1 -315.737,E2 -315.737} C_VEL
LIN {X 0,Y 608.433,Z 262.316,A -85,B 0,C 180,E1 -317.936,E2 -317.936} C_VEL
LIN {X 0,Y 608.441,Z 262.316,A -85,B 0,C 180,E1 -320.704,E2 -320.704} C_VEL
LIN {X 0,Y 608.457,Z 262.321,A -85,B 0,C 180,E1 -323.085,E2 -323.085} C_VEL
LIN {X 0,Y 608.455,Z 262.316,A -85,B 0,C 180,E1 -325.53,E2 -325.53} C_VEL
LIN {X 0,Y 608.436,Z 262.315,A -85,B 0,C 180,E1 -327.904,E2 -327.904} C_VEL
LIN {X 0,Y 608.439,Z 262.314,A -85,B 0,C 180,E1 -330.219,E2 -330.219} C_VEL
LIN {X 0,Y 608.484,Z 262.315,A -85,B 0,C 180,E1 -332.789,E2 -332.789} C_VEL
LIN {X 0,Y 608.432,Z 262.319,A -85,B 0,C 180,E1 -335.428,E2 -335.428} C_VEL
LIN {X 0,Y 608.453,Z 262.313,A -85,B 0,C 180,E1 -338.308,E2 -338.308} C_VEL
LIN {X 0,Y 608.444,Z 262.318,A -85,B 0,C 180,E1 -341.287,E2 -341.287} C_VEL
LIN {X 0,Y 608.418,Z 262.317,A -85,B 0,C 180,E1 -343.905,E2 -343.905} C_VEL
LIN {X 0,Y 608.461,Z 262.318,A -85,B 0,C 180,E1 -346.643,E2 -346.643} C_VEL
LIN {X 0,Y 608.423,Z 262.318,A -85,B 0,C 180,E1 -349.349,E2 -349.349} C_VEL
LIN {X 0,Y 608.413,Z 262.319,A -85,B 0,C 180,E1 -351.363,E2 -351.363} C_VEL
LIN {X 0,Y 608.422,Z 262.318,A -85,B 0,C 180,E1 -353.401,E2 -353.401} C_VEL
LIN {X 0,Y 608.401,Z 262.32,A -85,B 0,C 180,E1 -355.362,E2 -355.362} C_VEL
LIN {X 0,Y 608.427,Z 262.317,A -85,B 0,C 180,E1 -357.352,E2 -357.352} C_VEL
LIN {X 0,Y 608.428,Z 262.316,A -85,B 0,C 180,E1 -359.338,E2 -359.338} C_VEL
LIN {X 0,Y 608.416,Z 262.318,A -85,B 0,C 180,E1 -361.324,E2 -361.324} C_VEL
LIN {X 0,Y 608.397,Z 262.32,A -85,B 0,C 180,E1 -363.311,E2 -363.311} C_VEL
LIN {X 0,Y 608.408,Z 262.319,A -85,B 0,C 180,E1 -365.302,E2 -365.302} C_VEL
LIN {X 0,Y 608.4,Z 262.32,A -85,B 0,C 180,E1 -367.3,E2 -367.3} C_VEL
LIN {X 0,Y 608.411,Z 262.318,A -85,B 0,C 180,E1 -369.307,E2 -369.307} C_VEL
LIN {X 0,Y 608.398,Z 262.319,A -85,B 0,C 180,E1 -371.325,E2 -371.325} C_VEL
LIN {X 0,Y 608.402,Z 262.319,A -85,B 0,C 180,E1 -373.358,E2 -373.358} C_VEL
LIN {X 0,Y 608.409,Z 262.318,A -85,B 0,C 180,E1 -375.407,E2 -375.407} C_VEL
LIN {X 0,Y 608.392,Z 262.32,A -85,B 0,C 180,E1 -377.478,E2 -377.478} C_VEL
LIN {X 0,Y 608.437,Z 262.323,A -85,B 0,C 180,E1 -380.275,E2 -380.275} C_VEL
LIN {X 0,Y 608.397,Z 262.32,A -85,B 0,C 180,E1 -383.126,E2 -383.126} C_VEL
LIN {X 0,Y 608.419,Z 262.318,A -85,B 0,C 180,E1 -385.714,E2 -385.714} C_VEL
LIN {X 0,Y 608.455,Z 262.317,A -85,B 0,C 180,E1 -388.62,E2 -388.62} C_VEL
LIN {X 0,Y 608.414,Z 262.317,A -85,B 0,C 180,E1 -391.319,E2 -391.319} C_VEL
LIN {X 0,Y 608.411,Z 262.321,A -85,B 0,C 180,E1 -393.729,E2 -393.729} C_VEL
LIN {X 0,Y 608.432,Z 262.325,A -85,B 0,C 180,E1 -396.093,E2 -396.093} C_VEL
LIN {X 0,Y 608.407,Z 262.321,A -85,B 0,C 180,E1 -398.593,E2 -398.593} C_VEL
LIN {X 0,Y 608.41,Z 262.318,A -85,B 0,C 180,E1 -401.338,E2 -401.338} C_VEL
LIN {X 0,Y 608.461,Z 262.319,A -85,B 0,C 180,E1 -403.87,E2 -403.87} C_VEL
LIN {X 0,Y 608.434,Z 262.316,A -85,B 0,C 180,E1 -406.695,E2 -406.695} C_VEL
LIN {X 0,Y 608.409,Z 262.318,A -85,B 0,C 180,E1 -408.821,E2 -408.821} C_VEL
LIN {X 0,Y 608.459,Z 262.319,A -85,B 0,C 180,E1 -411.761,E2 -411.761} C_VEL
LIN {X 0,Y 608.419,Z 262.317,A -85,B 0,C 180,E1 -414.722,E2 -414.722} C_VEL
LIN {X 0,Y 608.427,Z 262.316,A -85,B 0,C 180,E1 -417.12,E2 -417.12} C_VEL
LIN {X 0,Y 608.476,Z 262.317,A -85,B 0,C 180,E1 -420.027,E2 -420.027} C_VEL
LIN {X 0,Y 608.421,Z 262.317,A -85,B 0,C 180,E1 -422.803,E2 -422.803} C_VEL
LIN {X 0,Y 608.448,Z 262.454,A -85,B 0,C 180,E1 -424.745,E2 -424.745} C_VEL
LIN {X 0,Y 608.665,Z 274.548,A -85,B 0,C 180,E1 -426.164,E2 -426.164} C_VEL
LIN {X 0,Y 608.595,Z 297.958,A -85,B 0,C 180,E1 -428.847,E2 -428.847} C_VEL
LIN {X 0,Y 608.574,Z 322.06,A -85,B 0,C 180,E1 -431.548,E2 -431.548} C_VEL
LIN {X 0,Y 608.727,Z 425.956,A -85,B 0,C 180,E1 -432.814,E2 -432.814} C_VEL
LIN {X 0,Y 608.682,Z 488.129,A -85,B 0,C 180,E1 -433.581,E2 -433.581} C_VEL
LIN {X 0,Y 608.65,Z 503.73,A -85,B 0,C 180,E1 -433.912,E2 -433.912} C_VEL
LIN {X 0,Y 608.618,Z 519.062,A -85,B 0,C 180,E1 -434.384,E2 -434.384} C_VEL
LIN {X 0,Y 608.606,Z 532.767,A -85,B 0,C 180,E1 -434.941,E2 -434.941} C_VEL
LIN {X 0,Y 608.575,Z 546.244,A -85,B 0,C 180,E1 -435.625,E2 -435.625} C_VEL
LIN {X 0,Y 608.554,Z 558.67,A -85,B 0,C 180,E1 -436.391,E2 -436.391} C_VEL
LIN {X 0,Y 608.528,Z 571.288,A -85,B 0,C 180,E1 -437.325,E2 -437.325} C_VEL
LIN {X 0,Y 608.496,Z 582.751,A -85,B 0,C 180,E1 -438.339,E2 -438.339} C_VEL
LIN {X 0,Y 608.476,Z 592.391,A -85,B 0,C 180,E1 -439.351,E2 -439.351} C_VEL
LIN {X 0,Y 608.477,Z 601.856,A -85,B 0,C 180,E1 -440.527,E2 -440.527} C_VEL
LIN {X 0,Y 608.455,Z 609.731,A -85,B 0,C 180,E1 -441.699,E2 -441.699} C_VEL
LIN {X 0,Y 608.441,Z 617.088,A -85,B 0,C 180,E1 -443.034,E2 -443.034} C_VEL
LIN {X 0,Y 608.449,Z 622.924,A -85,B 0,C 180,E1 -444.366,E2 -444.366} C_VEL
LIN {X 0,Y 608.427,Z 626.383,A -85,B 0,C 180,E1 -445.362,E2 -445.362} C_VEL
LIN {X 0,Y 608.421,Z 629.886,A -85,B 0,C 180,E1 -446.689,E2 -446.689} C_VEL
LIN {X 0,Y 608.442,Z 632.191,A -85,B 0,C 180,E1 -448.014,E2 -448.014} C_VEL
LIN {X 0,Y 608.436,Z 633.351,A -85,B 0,C 180,E1 -449.338,E2 -449.338} C_VEL
LIN {X 0,Y 608.436,Z 633.351,A -85,B 0,C 180,E1 -450.662,E2 -450.662} C_VEL
LIN {X 0,Y 608.442,Z 632.191,A -85,B 0,C 180,E1 -451.986,E2 -451.986} C_VEL
LIN {X 0,Y 608.421,Z 629.886,A -85,B 0,C 180,E1 -453.311,E2 -453.311} C_VEL
LIN {X 0,Y 608.427,Z 626.383,A -85,B 0,C 180,E1 -454.638,E2 -454.638} C_VEL
LIN {X 0,Y 608.431,Z 621.608,A -85,B 0,C 180,E1 -455.967,E2 -455.967} C_VEL
LIN {X 0,Y 608.458,Z 615.427,A -85,B 0,C 180,E1 -457.299,E2 -457.299} C_VEL
LIN {X 0,Y 608.465,Z 607.655,A -85,B 0,C 180,E1 -458.636,E2 -458.636} C_VEL
LIN {X 0,Y 608.471,Z 599.372,A -85,B 0,C 180,E1 -459.809,E2 -459.809} C_VEL
LIN {X 0,Y 608.492,Z 588.651,A -85,B 0,C 180,E1 -461.063,E2 -461.063} C_VEL
LIN {X 0,Y 608.522,Z 577.278,A -85,B 0,C 180,E1 -462.167,E2 -462.167} C_VEL
LIN {X 0,Y 608.548,Z 565.859,A -85,B 0,C 180,E1 -463.099,E2 -463.099} C_VEL
LIN {X 0,Y 608.562,Z 553.453,A -85,B 0,C 180,E1 -463.95,E2 -463.95} C_VEL
LIN {X 0,Y 608.569,Z 539.867,A -85,B 0,C 180,E1 -464.718,E2 -464.718} C_VEL
LIN {X 0,Y 608.633,Z 525.803,A -85,B 0,C 180,E1 -465.358,E2 -465.358} C_VEL
LIN {X 0,Y 608.636,Z 511.316,A -85,B 0,C 180,E1 -465.874,E2 -465.874} C_VEL
LIN {X 0,Y 608.689,Z 496.013,A -85,B 0,C 180,E1 -466.27,E2 -466.27} C_VEL
LIN {X 0,Y 608.687,Z 480.029,A -85,B 0,C 180,E1 -466.535,E2 -466.535} C_VEL
LIN {X 0,Y 608.683,Z 322.69,A -85,B 0,C 180,E1 -468.441,E2 -468.441} C_VEL
LIN {X 0,Y 608.541,Z 321.571,A -85,B 0,C 180,E1 -468.494,E2 -468.494} C_VEL
LIN {X 0,Y 608.619,Z 296.397,A -85,B 0,C 180,E1 -471.33,E2 -471.33} C_VEL
LIN {X 0,Y 608.682,Z 271.445,A -85,B 0,C 180,E1 -474.195,E2 -474.195} C_VEL
LIN {X 0,Y 608.448,Z 262.454,A -85,B 0,C 180,E1 -475.255,E2 -475.255} C_VEL
LIN {X 0,Y 608.442,Z 262.324,A -85,B 0,C 180,E1 -478.266,E2 -478.266} C_VEL
LIN {X 0,Y 608.453,Z 262.317,A -85,B 0,C 180,E1 -480.545,E2 -480.545} C_VEL
LIN {X 0,Y 608.427,Z 262.316,A -85,B 0,C 180,E1 -482.88,E2 -482.88} C_VEL
LIN {X 0,Y 608.419,Z 262.317,A -85,B 0,C 180,E1 -485.278,E2 -485.278} C_VEL
LIN {X 0,Y 608.462,Z 262.319,A -85,B 0,C 180,E1 -488.24,E2 -488.24} C_VEL
LIN {X 0,Y 608.41,Z 262.318,A -85,B 0,C 180,E1 -491.179,E2 -491.179} C_VEL
LIN {X 0,Y 608.465,Z 262.319,A -85,B 0,C 180,E1 -493.868,E2 -493.868} C_VEL
LIN {X 0,Y 608.424,Z 262.317,A -85,B 0,C 180,E1 -496.694,E2 -496.694} C_VEL
LIN {X 0,Y 608.398,Z 262.319,A -85,B 0,C 180,E1 -498.819,E2 -498.819} C_VEL
LIN {X 0,Y 608.457,Z 262.32,A -85,B 0,C 180,E1 -501.759,E2 -501.759} C_VEL
LIN {X 0,Y 608.398,Z 262.319,A -85,B 0,C 180,E1 -504.719,E2 -504.719} C_VEL
LIN {X 0,Y 608.452,Z 262.317,A -85,B 0,C 180,E1 -507.477,E2 -507.477} C_VEL
LIN {X 0,Y 608.43,Z 262.319,A -85,B 0,C 180,E1 -510.219,E2 -510.219} C_VEL
LIN {X 0,Y 608.402,Z 262.319,A -85,B 0,C 180,E1 -512.804,E2 -512.804} C_VEL
LIN {X 0,Y 608.428,Z 262.321,A -85,B 0,C 180,E1 -515.428,E2 -515.428} C_VEL
LIN {X 0,Y 608.42,Z 262.318,A -85,B 0,C 180,E1 -518.307,E2 -518.307} C_VEL
LIN {X 0,Y 608.397,Z 262.319,A -85,B 0,C 180,E1 -520.428,E2 -520.428} C_VEL
LIN {X 0,Y 608.465,Z 262.319,A -85,B 0,C 180,E1 -523.467,E2 -523.467} C_VEL
LIN {X 0,Y 608.414,Z 262.321,A -85,B 0,C 180,E1 -525.998,E2 -525.998} C_VEL
LIN {X 0,Y 608.416,Z 262.32,A -85,B 0,C 180,E1 -527.999,E2 -527.999} C_VEL
LIN {X 0,Y 608.408,Z 262.32,A -85,B 0,C 180,E1 -530.022,E2 -530.022} C_VEL
LIN {X 0,Y 608.401,Z 262.321,A -85,B 0,C 180,E1 -532.032,E2 -532.032} C_VEL
LIN {X 0,Y 608.412,Z 262.319,A -85,B 0,C 180,E1 -534.033,E2 -534.033} C_VEL
LIN {X 0,Y 608.404,Z 262.32,A -85,B 0,C 180,E1 -536.026,E2 -536.026} C_VEL
LIN {X 0,Y 608.408,Z 262.319,A -85,B 0,C 180,E1 -538.014,E2 -538.014} C_VEL
LIN {X 0,Y 608.431,Z 262.317,A -85,B 0,C 180,E1 -540,E2 -540} C_VEL
LIN {X 0,Y 608.411,Z 262.319,A -85,B 0,C 180,E1 -541.986,E2 -541.986} C_VEL
LIN {X 0,Y 608.408,Z 262.319,A -85,B 0,C 180,E1 -543.974,E2 -543.974} C_VEL
LIN {X 0,Y 608.418,Z 262.318,A -85,B 0,C 180,E1 -545.967,E2 -545.967} C_VEL
LIN {X 0,Y 608.41,Z 262.319,A -85,B 0,C 180,E1 -547.968,E2 -547.968} C_VEL
LIN {X 0,Y 608.452,Z 262.32,A -85,B 0,C 180,E1 -549.423,E2 -549.423} C_VEL
LIN {X 0,Y 607.748,Z 262.403,A -85,B 0,C 180,E1 -549.976,E2 -549.976} C_VEL
LIN {X 0,Y 604.885,Z 262.761,A -85,B 0,C 180,E1 -550.872,E2 -550.872} C_VEL
LIN {X 0,Y 602.485,Z 263.06,A -85,B 0,C 180,E1 -551.594,E2 -551.594} C_VEL
LIN {X 0,Y 601.452,Z 263.185,A -85,B 0,C 180,E1 -552.15,E2 -552.15} C_VEL
LIN {X 0,Y 601.366,Z 263.195,A -85,B 0,C 180,E1 -552.339,E2 -552.339} C_VEL
LIN {X 0,Y 601.387,Z 263.198,A -85,B 0,C 180,E1 -554.898,E2 -554.898} C_VEL
LIN {X 0,Y 601.378,Z 263.196,A -85,B 0,C 180,E1 -557.689,E2 -557.689} C_VEL
LIN {X 0,Y 601.392,Z 263.193,A -85,B 0,C 180,E1 -560.523,E2 -560.523} C_VEL
LIN {X 0,Y 601.377,Z 263.198,A -85,B 0,C 180,E1 -563.412,E2 -563.412} C_VEL
LIN {X 0,Y 601.385,Z 263.193,A -85,B 0,C 180,E1 -565.865,E2 -565.865} C_VEL
LIN {X 0,Y 601.379,Z 263.193,A -85,B 0,C 180,E1 -567.87,E2 -567.87} C_VEL
LIN {X 0,Y 601.387,Z 263.193,A -85,B 0,C 180,E1 -570.166,E2 -570.166} C_VEL
LIN {X 0,Y 601.398,Z 263.198,A -85,B 0,C 180,E1 -572.714,E2 -572.714} C_VEL
LIN {X 0,Y 601.402,Z 263.198,A -85,B 0,C 180,E1 -575.115,E2 -575.115} C_VEL
LIN {X 0,Y 601.426,Z 263.19,A -85,B 0,C 180,E1 -577.42,E2 -577.42} C_VEL
LIN {X 0,Y 601.392,Z 263.192,A -85,B 0,C 180,E1 -579.997,E2 -579.997} C_VEL
LIN {X 0,Y 601.402,Z 263.199,A -85,B 0,C 180,E1 -582.671,E2 -582.671} C_VEL
LIN {X 0,Y 601.391,Z 263.193,A -85,B 0,C 180,E1 -585.48,E2 -585.48} C_VEL
LIN {X 0,Y 601.413,Z 263.195,A -85,B 0,C 180,E1 -588.408,E2 -588.408} C_VEL
LIN {X 0,Y 601.404,Z 263.198,A -85,B 0,C 180,E1 -590.874,E2 -590.874} C_VEL
LIN {X 0,Y 601.399,Z 263.192,A -85,B 0,C 180,E1 -593.418,E2 -593.418} C_VEL
LIN {X 0,Y 601.412,Z 263.192,A -85,B 0,C 180,E1 -596.068,E2 -596.068} C_VEL
LIN {X 0,Y 601.437,Z 263.196,A -85,B 0,C 180,E1 -598.543,E2 -598.543} C_VEL
LIN {X 0,Y 601.42,Z 263.189,A -85,B 0,C 180,E1 -601.373,E2 -601.373} C_VEL
LIN {X 0,Y 601.393,Z 263.192,A -85,B 0,C 180,E1 -603.637,E2 -603.637} C_VEL
LIN {X 0,Y 601.414,Z 263.199,A -85,B 0,C 180,E1 -606.59,E2 -606.59} C_VEL
LIN {X 0,Y 601.409,Z 263.199,A -85,B 0,C 180,E1 -607.433,E2 -607.433} C_VEL
LIN {X 0,Y 601.671,Z 269.085,A -85,B 0,C 180,E1 -608.232,E2 -608.232} C_VEL
LIN {X 0,Y 601.597,Z 289.326,A -85,B 0,C 180,E1 -610.908,E2 -610.908} C_VEL
LIN {X 0,Y 601.575,Z 292.864,A -85,B 0,C 180,E1 -611.37,E2 -611.37} C_VEL
LIN {X 0,Y 601.993,Z 296.927,A -85,B 0,C 180,E1 -611.443,E2 -611.443} C_VEL
LIN {X 0,Y 601.88,Z 457.986,A -85,B 0,C 180,E1 -613.433,E2 -613.433} C_VEL
LIN {X 0,Y 601.824,Z 473.679,A -85,B 0,C 180,E1 -613.768,E2 -613.768} C_VEL
LIN {X 0,Y 601.753,Z 489.021,A -85,B 0,C 180,E1 -614.244,E2 -614.244} C_VEL
LIN {X 0,Y 601.725,Z 503.694,A -85,B 0,C 180,E1 -614.851,E2 -614.851} C_VEL
LIN {X 0,Y 601.658,Z 516.991,A -85,B 0,C 180,E1 -615.542,E2 -615.542} C_VEL
LIN {X 0,Y 601.604,Z 529.806,A -85,B 0,C 180,E1 -616.352,E2 -616.352} C_VEL
LIN {X 0,Y 601.541,Z 541.794,A -85,B 0,C 180,E1 -617.261,E2 -617.261} C_VEL
LIN {X 0,Y 601.489,Z 552.284,A -85,B 0,C 180,E1 -618.202,E2 -618.202} C_VEL
LIN {X 0,Y 601.43,Z 561.998,A -85,B 0,C 180,E1 -619.224,E2 -619.224} C_VEL
LIN {X 0,Y 601.428,Z 571.528,A -85,B 0,C 180,E1 -620.415,E2 -620.415} C_VEL
LIN {X 0,Y 601.378,Z 579.462,A -85,B 0,C 180,E1 -621.6,E2 -621.6} C_VEL
LIN {X 0,Y 601.368,Z 586.873,A -85,B 0,C 180,E1 -622.952,E2 -622.952} C_VEL
LIN {X 0,Y 601.372,Z 592.759,A -85,B 0,C 180,E1 -624.299,E2 -624.299} C_VEL
LIN {X 0,Y 601.329,Z 596.242,A -85,B 0,C 180,E1 -625.307,E2 -625.307} C_VEL
LIN {X 0,Y 601.336,Z 599.79,A -85,B 0,C 180,E1 -626.65,E2 -626.65} C_VEL
LIN {X 0,Y 601.342,Z 602.139,A -85,B 0,C 180,E1 -627.991,E2 -627.991} C_VEL
LIN {X 0,Y 601.334,Z 603.337,A -85,B 0,C 180,E1 -629.33,E2 -629.33} C_VEL
LIN {X 0,Y 601.336,Z 603.361,A -85,B 0,C 180,E1 -630.67,E2 -630.67} C_VEL
LIN {X 0,Y 601.343,Z 602.245,A -85,B 0,C 180,E1 -632.009,E2 -632.009} C_VEL
LIN {X 0,Y 601.339,Z 599.983,A -85,B 0,C 180,E1 -633.35,E2 -633.35} C_VEL
LIN {X 0,Y 601.329,Z 596.526,A -85,B 0,C 180,E1 -634.693,E2 -634.693} C_VEL
LIN {X 0,Y 601.357,Z 591.798,A -85,B 0,C 180,E1 -636.037,E2 -636.037} C_VEL
LIN {X 0,Y 601.364,Z 585.667,A -85,B 0,C 180,E1 -637.386,E2 -637.386} C_VEL
LIN {X 0,Y 601.387,Z 577.952,A -85,B 0,C 180,E1 -638.738,E2 -638.738} C_VEL
LIN {X 0,Y 601.428,Z 569.709,A -85,B 0,C 180,E1 -639.925,E2 -639.925} C_VEL
LIN {X 0,Y 601.443,Z 559.366,A -85,B 0,C 180,E1 -641.164,E2 -641.164} C_VEL
LIN {X 0,Y 601.503,Z 547.788,A -85,B 0,C 180,E1 -642.312,E2 -642.312} C_VEL
LIN {X 0,Y 601.557,Z 536.468,A -85,B 0,C 180,E1 -643.254,E2 -643.254} C_VEL
LIN {X 0,Y 601.623,Z 523.32,A -85,B 0,C 180,E1 -644.167,E2 -644.167} C_VEL
LIN {X 0,Y 601.661,Z 510.767,A -85,B 0,C 180,E1 -644.891,E2 -644.891} C_VEL
LIN {X 0,Y 601.765,Z 495.845,A -85,B 0,C 180,E1 -645.582,E2 -645.582} C_VEL
LIN {X 0,Y 601.816,Z 481.359,A -85,B 0,C 180,E1 -646.102,E2 -646.102} C_VEL
LIN {X 0,Y 601.874,Z 466.062,A -85,B 0,C 180,E1 -646.503,E2 -646.503} C_VEL
LIN {X 0,Y 601.893,Z 450.207,A -85,B 0,C 180,E1 -646.769,E2 -646.769} C_VEL
LIN {X 0,Y 601.934,Z 294.767,A -85,B 0,C 180,E1 -648.675,E2 -648.675} C_VEL
LIN {X 0,Y 601.548,Z 292.826,A -85,B 0,C 180,E1 -648.725,E2 -648.725} C_VEL
LIN {X 0,Y 601.652,Z 272.46,A -85,B 0,C 180,E1 -651.409,E2 -651.409} C_VEL
LIN {X 0,Y 601.446,Z 263.242,A -85,B 0,C 180,E1 -652.65,E2 -652.65} C_VEL
LIN {X 0,Y 601.401,Z 263.193,A -85,B 0,C 180,E1 -654.878,E2 -654.878} C_VEL
LIN {X 0,Y 601.414,Z 263.197,A -85,B 0,C 180,E1 -657.362,E2 -657.362} C_VEL
LIN {X 0,Y 601.415,Z 263.198,A -85,B 0,C 180,E1 -659.392,E2 -659.392} C_VEL
LIN {X 0,Y 601.405,Z 263.197,A -85,B 0,C 180,E1 -661.726,E2 -661.726} C_VEL
LIN {X 0,Y 601.424,Z 263.189,A -85,B 0,C 180,E1 -664.118,E2 -664.118} C_VEL
LIN {X 0,Y 601.433,Z 263.198,A -85,B 0,C 180,E1 -667.381,E2 -667.381} C_VEL
LIN {X 0,Y 601.404,Z 263.192,A -85,B 0,C 180,E1 -669.994,E2 -669.994} C_VEL
LIN {X 0,Y 601.402,Z 263.192,A -85,B 0,C 180,E1 -672.67,E2 -672.67} C_VEL
LIN {X 0,Y 601.391,Z 263.199,A -85,B 0,C 180,E1 -675.479,E2 -675.479} C_VEL
LIN {X 0,Y 601.413,Z 263.189,A -85,B 0,C 180,E1 -678.406,E2 -678.406} C_VEL
LIN {X 0,Y 601.403,Z 263.195,A -85,B 0,C 180,E1 -680.873,E2 -680.873} C_VEL
LIN {X 0,Y 601.397,Z 263.197,A -85,B 0,C 180,E1 -683.416,E2 -683.416} C_VEL
LIN {X 0,Y 601.405,Z 263.19,A -85,B 0,C 180,E1 -686.066,E2 -686.066} C_VEL
LIN {X 0,Y 601.43,Z 263.189,A -85,B 0,C 180,E1 -688.541,E2 -688.541} C_VEL
LIN {X 0,Y 601.41,Z 263.195,A -85,B 0,C 180,E1 -691.372,E2 -691.372} C_VEL
LIN {X 0,Y 601.382,Z 263.195,A -85,B 0,C 180,E1 -693.635,E2 -693.635} C_VEL
LIN {X 0,Y 601.401,Z 263.195,A -85,B 0,C 180,E1 -696.589,E2 -696.589} C_VEL
LIN {X 0,Y 601.398,Z 263.194,A -85,B 0,C 180,E1 -699.477,E2 -699.477} C_VEL
LIN {X 0,Y 601.379,Z 263.195,A -85,B 0,C 180,E1 -702.311,E2 -702.311} C_VEL
LIN {X 0,Y 601.39,Z 263.199,A -85,B 0,C 180,E1 -705.102,E2 -705.102} C_VEL
LIN {X 0,Y 601.385,Z 263.193,A -85,B 0,C 180,E1 -707.857,E2 -707.857} C_VEL
LIN {X 0,Y 601.41,Z 263.197,A -85,B 0,C 180,E1 -710.584,E2 -710.584} C_VEL
LIN {X 0,Y 601.375,Z 263.196,A -85,B 0,C 180,E1 -713.378,E2 -713.378} C_VEL
LIN {X 0,Y 601.376,Z 263.195,A -85,B 0,C 180,E1 -715.308,E2 -715.308} C_VEL
LIN {X 0,Y 601.397,Z 263.193,A -85,B 0,C 180,E1 -717.321,E2 -717.321} C_VEL
LIN {X 0,Y 601.404,Z 263.191,A -85,B 0,C 180,E1 -720,E2 -720} C_VEL
LIN {X 0,Y 601.438,Z 263.196,A -85,B 0,C 180,E1 -722.679,E2 -722.679} C_VEL
LIN {X 0,Y 601.374,Z 263.195,A -85,B 0,C 180,E1 -725.364,E2 -725.364} C_VEL
LIN {X 0,Y 601.353,Z 263.197,A -85,B 0,C 180,E1 -727.386,E2 -727.386} C_VEL
LIN {X 0,Y 601.376,Z 263.197,A -85,B 0,C 180,E1 -730.096,E2 -730.096} C_VEL
LIN {X 0,Y 601.39,Z 263.197,A -85,B 0,C 180,E1 -732.829,E2 -732.829} C_VEL
LIN {X 0,Y 601.361,Z 263.196,A -85,B 0,C 180,E1 -735.593,E2 -735.593} C_VEL
LIN {X 0,Y 601.346,Z 263.198,A -85,B 0,C 180,E1 -737.69,E2 -737.69} C_VEL
LIN {X 0,Y 601.41,Z 263.198,A -85,B 0,C 180,E1 -740.522,E2 -740.522} C_VEL
LIN {X 0,Y 601.351,Z 263.197,A -85,B 0,C 180,E1 -743.413,E2 -743.413} C_VEL
LIN {X 0,Y 601.37,Z 263.198,A -85,B 0,C 180,E1 -745.862,E2 -745.862} C_VEL
LIN {X 0,Y 601.405,Z 263.193,A -85,B 0,C 180,E1 -748.786,E2 -748.786} C_VEL
LIN {X 0,Y 601.383,Z 263.196,A -85,B 0,C 180,E1 -751.728,E2 -751.728} C_VEL
LIN {X 0,Y 601.394,Z 263.201,A -85,B 0,C 180,E1 -754.121,E2 -754.121} C_VEL
LIN {X 0,Y 601.366,Z 263.199,A -85,B 0,C 180,E1 -756.585,E2 -756.585} C_VEL
LIN {X 0,Y 601.369,Z 263.195,A -85,B 0,C 180,E1 -759.13,E2 -759.13} C_VEL
LIN {X 0,Y 601.411,Z 263.194,A -85,B 0,C 180,E1 -761.766,E2 -761.766} C_VEL
LIN {X 0,Y 601.389,Z 263.195,A -85,B 0,C 180,E1 -764.533,E2 -764.533} C_VEL
LIN {X 0,Y 601.363,Z 263.197,A -85,B 0,C 180,E1 -767.414,E2 -767.414} C_VEL
LIN {X 0,Y 601.392,Z 263.202,A -85,B 0,C 180,E1 -770.005,E2 -770.005} C_VEL
LIN {X 0,Y 601.391,Z 263.193,A -85,B 0,C 180,E1 -772.623,E2 -772.623} C_VEL
LIN {X 0,Y 601.372,Z 263.195,A -85,B 0,C 180,E1 -775.066,E2 -775.066} C_VEL
LIN {X 0,Y 601.41,Z 263.194,A -85,B 0,C 180,E1 -777.484,E2 -777.484} C_VEL
LIN {X 0,Y 601.426,Z 263.198,A -85,B 0,C 180,E1 -779.852,E2 -779.852} C_VEL
LIN {X 0,Y 601.379,Z 263.195,A -85,B 0,C 180,E1 -782.644,E2 -782.644} C_VEL
LIN {X 0,Y 601.407,Z 263.234,A -85,B 0,C 180,E1 -784.521,E2 -784.521} C_VEL
LIN {X 0,Y 601.843,Z 266.745,A -85,B 0,C 180,E1 -784.957,E2 -784.957} C_VEL
LIN {X 0,Y 601.769,Z 289.077,A -85,B 0,C 180,E1 -787.569,E2 -787.569} C_VEL
LIN {X 0,Y 601.686,Z 313.564,A -85,B 0,C 180,E1 -790.379,E2 -790.379} C_VEL
LIN {X 0,Y 601.628,Z 321.873,A -85,B 0,C 180,E1 -791.32,E2 -791.32} C_VEL
LIN {X 0,Y 602.027,Z 326.059,A -85,B 0,C 180,E1 -791.389,E2 -791.389} C_VEL
LIN {X 0,Y 601.878,Z 488.493,A -85,B 0,C 180,E1 -793.396,E2 -793.396} C_VEL
LIN {X 0,Y 601.829,Z 503.728,A -85,B 0,C 180,E1 -793.724,E2 -793.724} C_VEL
LIN {X 0,Y 601.767,Z 519.06,A -85,B 0,C 180,E1 -794.201,E2 -794.201} C_VEL
LIN {X 0,Y 601.719,Z 532.77,A -85,B 0,C 180,E1 -794.764,E2 -794.764} C_VEL
LIN {X 0,Y 601.661,Z 546.241,A -85,B 0,C 180,E1 -795.455,E2 -795.455} C_VEL
LIN {X 0,Y 601.617,Z 559.453,A -85,B 0,C 180,E1 -796.283,E2 -796.283} C_VEL
LIN {X 0,Y 601.532,Z 571.289,A -85,B 0,C 180,E1 -797.175,E2 -797.175} C_VEL
LIN {X 0,Y 601.487,Z 582.751,A -85,B 0,C 180,E1 -798.201,E2 -798.201} C_VEL
LIN {X 0,Y 601.431,Z 592.391,A -85,B 0,C 180,E1 -799.224,E2 -799.224} C_VEL
LIN {X 0,Y 601.428,Z 601.857,A -85,B 0,C 180,E1 -800.415,E2 -800.415} C_VEL
LIN {X 0,Y 601.368,Z 609.732,A -85,B 0,C 180,E1 -801.6,E2 -801.6} C_VEL
LIN {X 0,Y 601.368,Z 617.089,A -85,B 0,C 180,E1 -802.952,E2 -802.952} C_VEL
LIN {X 0,Y 601.371,Z 622.924,A -85,B 0,C 180,E1 -804.299,E2 -804.299} C_VEL
LIN {X 0,Y 601.33,Z 626.384,A -85,B 0,C 180,E1 -805.307,E2 -805.307} C_VEL
LIN {X 0,Y 601.337,Z 629.886,A -85,B 0,C 180,E1 -806.65,E2 -806.65} C_VEL
LIN {X 0,Y 601.341,Z 632.192,A -85,B 0,C 180,E1 -807.991,E2 -807.991} C_VEL
LIN {X 0,Y 601.337,Z 633.35,A -85,B 0,C 180,E1 -809.33,E2 -809.33} C_VEL
LIN {X 0,Y 601.337,Z 633.35,A -85,B 0,C 180,E1 -810.67,E2 -810.67} C_VEL
LIN {X 0,Y 601.341,Z 632.192,A -85,B 0,C 180,E1 -812.009,E2 -812.009} C_VEL
LIN {X 0,Y 601.337,Z 629.886,A -85,B 0,C 180,E1 -813.35,E2 -813.35} C_VEL
LIN {X 0,Y 601.33,Z 626.384,A -85,B 0,C 180,E1 -814.693,E2 -814.693} C_VEL
LIN {X 0,Y 601.352,Z 621.609,A -85,B 0,C 180,E1 -816.038,E2 -816.038} C_VEL
LIN {X 0,Y 601.366,Z 615.426,A -85,B 0,C 180,E1 -817.386,E2 -817.386} C_VEL
LIN {X 0,Y 601.387,Z 607.655,A -85,B 0,C 180,E1 -818.738,E2 -818.738} C_VEL
LIN {X 0,Y 601.427,Z 599.372,A -85,B 0,C 180,E1 -819.925,E2 -819.925} C_VEL
LIN {X 0,Y 601.46,Z 588.932,A -85,B 0,C 180,E1 -821.165,E2 -821.165} C_VEL
LIN {X 0,Y 601.513,Z 579.196,A -85,B 0,C 180,E1 -822.14,E2 -822.14} C_VEL
LIN {X 0,Y 601.57,Z 567.021,A -85,B 0,C 180,E1 -823.168,E2 -823.168} C_VEL
LIN {X 0,Y 601.605,Z 555.083,A -85,B 0,C 180,E1 -824.011,E2 -824.011} C_VEL
LIN {X 0,Y 601.668,Z 541.534,A -85,B 0,C 180,E1 -824.804,E2 -824.804} C_VEL
LIN {X 0,Y 601.765,Z 526.852,A -85,B 0,C 180,E1 -825.495,E2 -825.495} C_VEL
LIN {X 0,Y 601.788,Z 512.631,A -85,B 0,C 180,E1 -826.016,E2 -826.016} C_VEL
LIN {X 0,Y 601.859,Z 497.678,A -85,B 0,C 180,E1 -826.42,E2 -826.42} C_VEL
LIN {X 0,Y 601.869,Z 482.694,A -85,B 0,C 180,E1 -826.69,E2 -826.69} C_VEL
LIN {X 0,Y 601.904,Z 323.494,A -85,B 0,C 180,E1 -828.647,E2 -828.647} C_VEL
LIN {X 0,Y 601.627,Z 321.749,A -85,B 0,C 180,E1 -828.694,E2 -828.694} C_VEL
LIN {X 0,Y 601.749,Z 296.397,A -85,B 0,C 180,E1 -831.585,E2 -831.585} C_VEL
LIN {X 0,Y 601.875,Z 272.31,A -85,B 0,C 180,E1 -834.385,E2 -834.385} C_VEL
LIN {X 0,Y 601.82,Z 265.185,A -85,B 0,C 180,E1 -835.229,E2 -835.229} C_VEL
LIN {X 0,Y 601.414,Z 263.195,A -85,B 0,C 180,E1 -835.502,E2 -835.502} C_VEL
LIN {X 0,Y 601.408,Z 263.194,A -85,B 0,C 180,E1 -838.627,E2 -838.627} C_VEL
LIN {X 0,Y 601.397,Z 263.192,A -85,B 0,C 180,E1 -840.942,E2 -840.942} C_VEL
LIN {X 0,Y 601.403,Z 263.191,A -85,B 0,C 180,E1 -843.314,E2 -843.314} C_VEL
LIN {X 0,Y 601.395,Z 263.2,A -85,B 0,C 180,E1 -846.26,E2 -846.26} C_VEL
LIN {X 0,Y 601.38,Z 263.194,A -85,B 0,C 180,E1 -849.128,E2 -849.128} C_VEL
LIN {X 0,Y 601.413,Z 263.195,A -85,B 0,C 180,E1 -851.765,E2 -851.765} C_VEL
LIN {X 0,Y 601.389,Z 263.195,A -85,B 0,C 180,E1 -854.532,E2 -854.532} C_VEL
LIN {X 0,Y 601.399,Z 263.193,A -85,B 0,C 180,E1 -857.409,E2 -857.409} C_VEL
LIN {X 0,Y 601.386,Z 263.202,A -85,B 0,C 180,E1 -860.003,E2 -860.003} C_VEL
LIN {X 0,Y 601.38,Z 263.194,A -85,B 0,C 180,E1 -862.623,E2 -862.623} C_VEL
LIN {X 0,Y 601.366,Z 263.196,A -85,B 0,C 180,E1 -865.065,E2 -865.065} C_VEL
LIN {X 0,Y 601.42,Z 263.193,A -85,B 0,C 180,E1 -867.484,E2 -867.484} C_VEL
LIN {X 0,Y 601.393,Z 263.201,A -85,B 0,C 180,E1 -869.855,E2 -869.855} C_VEL
LIN {X 0,Y 601.379,Z 263.198,A -85,B 0,C 180,E1 -872.131,E2 -872.131} C_VEL
LIN {X 0,Y 601.366,Z 263.196,A -85,B 0,C 180,E1 -874.38,E2 -874.38} C_VEL
LIN {X 0,Y 601.354,Z 263.197,A -85,B 0,C 180,E1 -876.587,E2 -876.587} C_VEL
LIN {X 0,Y 601.411,Z 263.197,A -85,B 0,C 180,E1 -879.478,E2 -879.478} C_VEL
LIN {X 0,Y 601.347,Z 263.198,A -85,B 0,C 180,E1 -882.31,E2 -882.31} C_VEL
LIN {X 0,Y 601.359,Z 263.196,A -85,B 0,C 180,E1 -884.407,E2 -884.407} C_VEL
LIN {X 0,Y 601.385,Z 263.197,A -85,B 0,C 180,E1 -887.171,E2 -887.171} C_VEL
LIN {X 0,Y 601.374,Z 263.198,A -85,B 0,C 180,E1 -889.904,E2 -889.904} C_VEL
LIN {X 0,Y 601.351,Z 263.197,A -85,B 0,C 180,E1 -892.614,E2 -892.614} C_VEL
LIN {X 0,Y 601.419,Z 263.196,A -85,B 0,C 180,E1 -895.308,E2 -895.308} C_VEL
LIN {X 0,Y 601.382,Z 263.195,A -85,B 0,C 180,E1 -897.991,E2 -897.991} C_VEL
LIN {X 0,Y 601.402,Z 263.192,A -85,B 0,C 180,E1 -900,E2 -900} C_VEL
LIN {X 0,Y 601.393,Z 263.193,A -85,B 0,C 180,E1 -902.679,E2 -902.679} C_VEL
LIN {X 0,Y 601.422,Z 263.198,A -85,B 0,C 180,E1 -905.364,E2 -905.364} C_VEL
LIN {X 0,Y 601.383,Z 263.193,A -85,B 0,C 180,E1 -908.062,E2 -908.062} C_VEL
LIN {X 0,Y 601.379,Z 263.197,A -85,B 0,C 180,E1 -910.777,E2 -910.777} C_VEL
LIN {X 0,Y 601.366,Z 263.195,A -85,B 0,C 180,E1 -912.339,E2 -912.339} C_VEL
LIN {X 0,Y 600.694,Z 263.285,A -85,B 0,C 180,E1 -912.898,E2 -912.898} C_VEL
LIN {X 0,Y 597.848,Z 263.643,A -85,B 0,C 180,E1 -913.806,E2 -913.806} C_VEL
LIN {X 0,Y 595.448,Z 263.943,A -85,B 0,C 180,E1 -914.536,E2 -914.536} C_VEL
LIN {X 0,Y 594.417,Z 264.07,A -85,B 0,C 180,E1 -915.099,E2 -915.099} C_VEL
LIN {X 0,Y 594.332,Z 264.077,A -85,B 0,C 180,E1 -915.29,E2 -915.29} C_VEL
LIN {X 0,Y 594.325,Z 264.073,A -85,B 0,C 180,E1 -917.906,E2 -917.906} C_VEL
LIN {X 0,Y 594.374,Z 264.07,A -85,B 0,C 180,E1 -920.777,E2 -920.777} C_VEL
LIN {X 0,Y 594.341,Z 264.072,A -85,B 0,C 180,E1 -923.706,E2 -923.706} C_VEL
LIN {X 0,Y 594.362,Z 264.067,A -85,B 0,C 180,E1 -926.021,E2 -926.021} C_VEL
LIN {X 0,Y 594.352,Z 264.068,A -85,B 0,C 180,E1 -928.228,E2 -928.228} C_VEL
LIN {X 0,Y 594.361,Z 264.072,A -85,B 0,C 180,E1 -930.561,E2 -930.561} C_VEL
LIN {X 0,Y 594.363,Z 264.078,A -85,B 0,C 180,E1 -932.951,E2 -932.951} C_VEL
LIN {X 0,Y 594.344,Z 264.073,A -85,B 0,C 180,E1 -935.41,E2 -935.41} C_VEL
LIN {X 0,Y 594.365,Z 264.067,A -85,B 0,C 180,E1 -937.942,E2 -937.942} C_VEL
LIN {X 0,Y 594.368,Z 264.077,A -85,B 0,C 180,E1 -940.823,E2 -940.823} C_VEL
LIN {X 0,Y 594.359,Z 264.071,A -85,B 0,C 180,E1 -943.3,E2 -943.3} C_VEL
LIN {X 0,Y 594.353,Z 264.071,A -85,B 0,C 180,E1 -946.162,E2 -946.162} C_VEL
LIN {X 0,Y 594.37,Z 264.07,A -85,B 0,C 180,E1 -949.179,E2 -949.179} C_VEL
LIN {X 0,Y 594.37,Z 264.068,A -85,B 0,C 180,E1 -952.059,E2 -952.059} C_VEL
LIN {X 0,Y 594.357,Z 264.079,A -85,B 0,C 180,E1 -954.676,E2 -954.676} C_VEL
LIN {X 0,Y 594.373,Z 264.07,A -85,B 0,C 180,E1 -957.09,E2 -957.09} C_VEL
LIN {X 0,Y 594.365,Z 264.068,A -85,B 0,C 180,E1 -959.676,E2 -959.676} C_VEL
LIN {X 0,Y 594.373,Z 264.076,A -85,B 0,C 180,E1 -962.54,E2 -962.54} C_VEL
LIN {X 0,Y 594.374,Z 264.073,A -85,B 0,C 180,E1 -964.808,E2 -964.808} C_VEL
LIN {X 0,Y 594.371,Z 264.122,A -85,B 0,C 180,E1 -967.276,E2 -967.276} C_VEL
LIN {X 0,Y 594.754,Z 269.09,A -85,B 0,C 180,E1 -967.965,E2 -967.965} C_VEL
LIN {X 0,Y 594.667,Z 289.331,A -85,B 0,C 180,E1 -970.676,E2 -970.676} C_VEL
LIN {X 0,Y 594.617,Z 292.926,A -85,B 0,C 180,E1 -971.152,E2 -971.152} C_VEL
LIN {X 0,Y 595.268,Z 297.135,A -85,B 0,C 180,E1 -971.228,E2 -971.228} C_VEL
LIN {X 0,Y 595.09,Z 458.451,A -85,B 0,C 180,E1 -973.246,E2 -973.246} C_VEL
LIN {X 0,Y 595.017,Z 473.7,A -85,B 0,C 180,E1 -973.577,E2 -973.577} C_VEL
LIN {X 0,Y 594.911,Z 489.035,A -85,B 0,C 180,E1 -974.058,E2 -974.058} C_VEL
LIN {X 0,Y 594.857,Z 503.705,A -85,B 0,C 180,E1 -974.672,E2 -974.672} C_VEL
LIN {X 0,Y 594.743,Z 517.004,A -85,B 0,C 180,E1 -975.37,E2 -975.37} C_VEL
LIN {X 0,Y 594.67,Z 529.995,A -85,B 0,C 180,E1 -976.202,E2 -976.202} C_VEL
LIN {X 0,Y 594.552,Z 542.862,A -85,B 0,C 180,E1 -977.195,E2 -977.195} C_VEL
LIN {X 0,Y 594.468,Z 554.065,A -85,B 0,C 180,E1 -978.233,E2 -978.233} C_VEL
LIN {X 0,Y 594.412,Z 564.948,A -85,B 0,C 180,E1 -979.44,E2 -979.44} C_VEL
LIN {X 0,Y 594.357,Z 573.993,A -85,B 0,C 180,E1 -980.643,E2 -980.643} C_VEL
LIN {X 0,Y 594.325,Z 581.487,A -85,B 0,C 180,E1 -981.842,E2 -981.842} C_VEL
LIN {X 0,Y 594.277,Z 588.491,A -85,B 0,C 180,E1 -983.208,E2 -983.208} C_VEL
LIN {X 0,Y 594.273,Z 593.999,A -85,B 0,C 180,E1 -984.571,E2 -984.571} C_VEL
LIN {X 0,Y 594.254,Z 598.171,A -85,B 0,C 180,E1 -985.931,E2 -985.931} C_VEL
LIN {X 0,Y 594.221,Z 601.112,A -85,B 0,C 180,E1 -987.288,E2 -987.288} C_VEL
LIN {X 0,Y 594.244,Z 602.88,A -85,B 0,C 180,E1 -988.645,E2 -988.645} C_VEL
LIN {X 0,Y 594.234,Z 603.496,A -85,B 0,C 180,E1 -990,E2 -990} C_VEL
LIN {X 0,Y 594.246,Z 602.944,A -85,B 0,C 180,E1 -991.355,E2 -991.355} C_VEL
LIN {X 0,Y 594.224,Z 601.259,A -85,B 0,C 180,E1 -992.712,E2 -992.712} C_VEL
LIN {X 0,Y 594.254,Z 598.407,A -85,B 0,C 180,E1 -994.069,E2 -994.069} C_VEL
LIN {X 0,Y 594.273,Z 594.325,A -85,B 0,C 180,E1 -995.429,E2 -995.429} C_VEL
LIN {X 0,Y 594.277,Z 588.916,A -85,B 0,C 180,E1 -996.792,E2 -996.792} C_VEL
LIN {X 0,Y 594.324,Z 582.018,A -85,B 0,C 180,E1 -998.158,E2 -998.158} C_VEL
LIN {X 0,Y 594.339,Z 573.416,A -85,B 0,C 180,E1 -999.529,E2 -999.529} C_VEL
LIN {X 0,Y 594.401,Z 564.267,A -85,B 0,C 180,E1 -1000.732,E2 -1000.732} C_VEL
LIN {X 0,Y 594.466,Z 553.214,A -85,B 0,C 180,E1 -1001.94,E2 -1001.94} C_VEL
LIN {X 0,Y 594.56,Z 541.839,A -85,B 0,C 180,E1 -1002.978,E2 -1002.978} C_VEL
LIN {X 0,Y 594.66,Z 529.458,A -85,B 0,C 180,E1 -1003.925,E2 -1003.925} C_VEL
LIN {X 0,Y 594.724,Z 517.049,A -85,B 0,C 180,E1 -1004.718,E2 -1004.718} C_VEL
LIN {X 0,Y 594.857,Z 503.754,A -85,B 0,C 180,E1 -1005.416,E2 -1005.416} C_VEL
LIN {X 0,Y 594.914,Z 489.084,A -85,B 0,C 180,E1 -1006.029,E2 -1006.029} C_VEL
LIN {X 0,Y 595.035,Z 473.944,A -85,B 0,C 180,E1 -1006.506,E2 -1006.506} C_VEL
LIN {X 0,Y 595.084,Z 458.22,A -85,B 0,C 180,E1 -1006.849,E2 -1006.849} C_VEL
LIN {X 0,Y 595.287,Z 296.678,A -85,B 0,C 180,E1 -1008.867,E2 -1008.867} C_VEL
LIN {X 0,Y 594.624,Z 292.927,A -85,B 0,C 180,E1 -1008.938,E2 -1008.938} C_VEL
LIN {X 0,Y 594.764,Z 272.455,A -85,B 0,C 180,E1 -1011.67,E2 -1011.67} C_VEL
LIN {X 0,Y 594.728,Z 266.272,A -85,B 0,C 180,E1 -1012.508,E2 -1012.508} C_VEL
LIN {X 0,Y 594.371,Z 264.073,A -85,B 0,C 180,E1 -1012.852,E2 -1012.852} C_VEL
LIN {X 0,Y 594.377,Z 264.072,A -85,B 0,C 180,E1 -1015.192,E2 -1015.192} C_VEL
LIN {X 0,Y 594.384,Z 264.076,A -85,B 0,C 180,E1 -1017.526,E2 -1017.526} C_VEL
LIN {X 0,Y 594.368,Z 264.068,A -85,B 0,C 180,E1 -1020.325,E2 -1020.325} C_VEL
LIN {X 0,Y 594.374,Z 264.069,A -85,B 0,C 180,E1 -1022.949,E2 -1022.949} C_VEL
LIN {X 0,Y 594.375,Z 264.077,A -85,B 0,C 180,E1 -1025.406,E2 -1025.406} C_VEL
LIN {X 0,Y 594.373,Z 264.069,A -85,B 0,C 180,E1 -1027.94,E2 -1027.94} C_VEL
LIN {X 0,Y 594.372,Z 264.068,A -85,B 0,C 180,E1 -1030.821,E2 -1030.821} C_VEL
LIN {X 0,Y 594.353,Z 264.071,A -85,B 0,C 180,E1 -1033.838,E2 -1033.838} C_VEL
LIN {X 0,Y 594.359,Z 264.07,A -85,B 0,C 180,E1 -1036.7,E2 -1036.7} C_VEL
LIN {X 0,Y 594.355,Z 264.076,A -85,B 0,C 180,E1 -1039.432,E2 -1039.432} C_VEL
LIN {X 0,Y 594.378,Z 264.066,A -85,B 0,C 180,E1 -1042.391,E2 -1042.391} C_VEL
LIN {X 0,Y 594.385,Z 264.071,A -85,B 0,C 180,E1 -1045.42,E2 -1045.42} C_VEL
LIN {X 0,Y 594.377,Z 264.066,A -85,B 0,C 180,E1 -1048.355,E2 -1048.355} C_VEL
LIN {X 0,Y 594.369,Z 264.076,A -85,B 0,C 180,E1 -1051.042,E2 -1051.042} C_VEL
LIN {X 0,Y 594.374,Z 264.072,A -85,B 0,C 180,E1 -1053.3,E2 -1053.3} C_VEL
LIN {X 0,Y 594.356,Z 264.069,A -85,B 0,C 180,E1 -1056.294,E2 -1056.294} C_VEL
LIN {X 0,Y 594.379,Z 264.071,A -85,B 0,C 180,E1 -1059.223,E2 -1059.223} C_VEL
LIN {X 0,Y 594.327,Z 264.072,A -85,B 0,C 180,E1 -1062.094,E2 -1062.094} C_VEL
LIN {X 0,Y 594.345,Z 264.071,A -85,B 0,C 180,E1 -1064.218,E2 -1064.218} C_VEL
LIN {X 0,Y 594.344,Z 264.077,A -85,B 0,C 180,E1 -1067.016,E2 -1067.016} C_VEL
LIN {X 0,Y 594.347,Z 264.075,A -85,B 0,C 180,E1 -1069.094,E2 -1069.094} C_VEL
LIN {X 0,Y 594.337,Z 264.071,A -85,B 0,C 180,E1 -1071.842,E2 -1071.842} C_VEL
LIN {X 0,Y 594.385,Z 264.072,A -85,B 0,C 180,E1 -1074.572,E2 -1074.572} C_VEL
LIN {X 0,Y 594.367,Z 264.069,A -85,B 0,C 180,E1 -1077.289,E2 -1077.289} C_VEL
LIN {X 0,Y 594.375,Z 264.067,A -85,B 0,C 180,E1 -1080,E2 -1080} C_VEL
LIN {X 0,Y 594.399,Z 264.072,A -85,B 0,C 180,E1 -1082.711,E2 -1082.711} C_VEL
LIN {X 0,Y 594.341,Z 264.07,A -85,B 0,C 180,E1 -1085.428,E2 -1085.428} C_VEL
LIN {X 0,Y 594.326,Z 264.072,A -85,B 0,C 180,E1 -1087.474,E2 -1087.474} C_VEL
LIN {X 0,Y 594.313,Z 264.073,A -85,B 0,C 180,E1 -1089.529,E2 -1089.529} C_VEL
LIN {X 0,Y 594.359,Z 264.075,A -85,B 0,C 180,E1 -1092.289,E2 -1092.289} C_VEL
LIN {X 0,Y 594.341,Z 264.072,A -85,B 0,C 180,E1 -1095.079,E2 -1095.079} C_VEL
LIN {X 0,Y 594.32,Z 264.073,A -85,B 0,C 180,E1 -1097.195,E2 -1097.195} C_VEL
LIN {X 0,Y 594.342,Z 264.075,A -85,B 0,C 180,E1 -1100.055,E2 -1100.055} C_VEL
LIN {X 0,Y 594.331,Z 264.073,A -85,B 0,C 180,E1 -1102.969,E2 -1102.969} C_VEL
LIN {X 0,Y 594.306,Z 264.075,A -85,B 0,C 180,E1 -1105.196,E2 -1105.196} C_VEL
LIN {X 0,Y 594.329,Z 264.073,A -85,B 0,C 180,E1 -1107.519,E2 -1107.519} C_VEL
LIN {X 0,Y 594.356,Z 264.078,A -85,B 0,C 180,E1 -1110.326,E2 -1110.326} C_VEL
LIN {X 0,Y 594.362,Z 264.068,A -85,B 0,C 180,E1 -1112.951,E2 -1112.951} C_VEL
LIN {X 0,Y 594.304,Z 264.076,A -85,B 0,C 180,E1 -1115.412,E2 -1115.412} C_VEL
LIN {X 0,Y 594.359,Z 264.075,A -85,B 0,C 180,E1 -1117.943,E2 -1117.943} C_VEL
LIN {X 0,Y 594.348,Z 264.069,A -85,B 0,C 180,E1 -1120.821,E2 -1120.821} C_VEL
LIN {X 0,Y 594.339,Z 264.071,A -85,B 0,C 180,E1 -1123.302,E2 -1123.302} C_VEL
LIN {X 0,Y 594.336,Z 264.079,A -85,B 0,C 180,E1 -1126.164,E2 -1126.164} C_VEL
LIN {X 0,Y 594.361,Z 264.07,A -85,B 0,C 180,E1 -1128.536,E2 -1128.536} C_VEL
LIN {X 0,Y 594.359,Z 264.07,A -85,B 0,C 180,E1 -1131.299,E2 -1131.299} C_VEL
LIN {X 0,Y 594.349,Z 264.077,A -85,B 0,C 180,E1 -1133.757,E2 -1133.757} C_VEL
LIN {X 0,Y 594.366,Z 264.072,A -85,B 0,C 180,E1 -1136.239,E2 -1136.239} C_VEL
LIN {X 0,Y 594.356,Z 264.069,A -85,B 0,C 180,E1 -1138.65,E2 -1138.65} C_VEL
LIN {X 0,Y 594.37,Z 264.068,A -85,B 0,C 180,E1 -1141.044,E2 -1141.044} C_VEL
LIN {X 0,Y 594.379,Z 264.074,A -85,B 0,C 180,E1 -1144.245,E2 -1144.245} C_VEL
LIN {X 0,Y 594.432,Z 264.404,A -85,B 0,C 180,E1 -1144.341,E2 -1144.341} C_VEL
LIN {X 0,Y 595.046,Z 268.306,A -85,B 0,C 180,E1 -1144.838,E2 -1144.838} C_VEL
LIN {X 0,Y 594.908,Z 291.946,A -85,B 0,C 180,E1 -1147.633,E2 -1147.633} C_VEL
LIN {X 0,Y 594.759,Z 316.685,A -85,B 0,C 180,E1 -1150.5,E2 -1150.5} C_VEL
LIN {X 0,Y 594.7,Z 321.89,A -85,B 0,C 180,E1 -1151.096,E2 -1151.096} C_VEL
LIN {X 0,Y 595.312,Z 325.444,A -85,B 0,C 180,E1 -1151.163,E2 -1151.163} C_VEL
LIN {X 0,Y 595.085,Z 488.316,A -85,B 0,C 180,E1 -1153.198,E2 -1153.198} C_VEL
LIN {X 0,Y 595.025,Z 503.727,A -85,B 0,C 180,E1 -1153.533,E2 -1153.533} C_VEL
LIN {X 0,Y 594.932,Z 519.058,A -85,B 0,C 180,E1 -1154.015,E2 -1154.015} C_VEL
LIN {X 0,Y 594.857,Z 532.772,A -85,B 0,C 180,E1 -1154.584,E2 -1154.584} C_VEL
LIN {X 0,Y 594.737,Z 546.244,A -85,B 0,C 180,E1 -1155.282,E2 -1155.282} C_VEL
LIN {X 0,Y 594.68,Z 558.798,A -85,B 0,C 180,E1 -1156.076,E2 -1156.076} C_VEL
LIN {X 0,Y 594.56,Z 571.29,A -85,B 0,C 180,E1 -1157.022,E2 -1157.022} C_VEL
LIN {X 0,Y 594.465,Z 582.752,A -85,B 0,C 180,E1 -1158.06,E2 -1158.06} C_VEL
LIN {X 0,Y 594.389,Z 592.392,A -85,B 0,C 180,E1 -1159.095,E2 -1159.095} C_VEL
LIN {X 0,Y 594.366,Z 601.857,A -85,B 0,C 180,E1 -1160.3,E2 -1160.3} C_VEL
LIN {X 0,Y 594.31,Z 609.732,A -85,B 0,C 180,E1 -1161.5,E2 -1161.5} C_VEL
LIN {X 0,Y 594.292,Z 617.089,A -85,B 0,C 180,E1 -1162.867,E2 -1162.867} C_VEL
LIN {X 0,Y 594.296,Z 622.925,A -85,B 0,C 180,E1 -1164.231,E2 -1164.231} C_VEL
LIN {X 0,Y 594.232,Z 626.384,A -85,B 0,C 180,E1 -1165.251,E2 -1165.251} C_VEL
LIN {X 0,Y 594.256,Z 629.887,A -85,B 0,C 180,E1 -1166.61,E2 -1166.61} C_VEL
LIN {X 0,Y 594.24,Z 632.193,A -85,B 0,C 180,E1 -1167.967,E2 -1167.967} C_VEL
LIN {X 0,Y 594.237,Z 633.35,A -85,B 0,C 180,E1 -1169.322,E2 -1169.322} C_VEL
LIN {X 0,Y 594.237,Z 633.35,A -85,B 0,C 180,E1 -1170.678,E2 -1170.678} C_VEL
LIN {X 0,Y 594.24,Z 632.192,A -85,B 0,C 180,E1 -1172.033,E2 -1172.033} C_VEL
LIN {X 0,Y 594.256,Z 629.886,A -85,B 0,C 180,E1 -1173.39,E2 -1173.39} C_VEL
LIN {X 0,Y 594.232,Z 626.384,A -85,B 0,C 180,E1 -1174.749,E2 -1174.749} C_VEL
LIN {X 0,Y 594.275,Z 621.609,A -85,B 0,C 180,E1 -1176.11,E2 -1176.11} C_VEL
LIN {X 0,Y 594.287,Z 615.426,A -85,B 0,C 180,E1 -1177.474,E2 -1177.474} C_VEL
LIN {X 0,Y 594.331,Z 607.653,A -85,B 0,C 180,E1 -1178.843,E2 -1178.843} C_VEL
LIN {X 0,Y 594.387,Z 599.372,A -85,B 0,C 180,E1 -1180.044,E2 -1180.044} C_VEL
LIN {X 0,Y 594.433,Z 589.559,A -85,B 0,C 180,E1 -1181.231,E2 -1181.231} C_VEL
LIN {X 0,Y 594.53,Z 579.195,A -85,B 0,C 180,E1 -1182.285,E2 -1182.285} C_VEL
LIN {X 0,Y 594.581,Z 567.022,A -85,B 0,C 180,E1 -1183.326,E2 -1183.326} C_VEL
LIN {X 0,Y 594.693,Z 555.08,A -85,B 0,C 180,E1 -1184.177,E2 -1184.177} C_VEL
LIN {X 0,Y 594.782,Z 541.531,A -85,B 0,C 180,E1 -1184.979,E2 -1184.979} C_VEL
LIN {X 0,Y 594.905,Z 526.849,A -85,B 0,C 180,E1 -1185.678,E2 -1185.678} C_VEL
LIN {X 0,Y 594.967,Z 512.631,A -85,B 0,C 180,E1 -1186.204,E2 -1186.204} C_VEL
LIN {X 0,Y 595.051,Z 498.12,A -85,B 0,C 180,E1 -1186.603,E2 -1186.603} C_VEL
LIN {X 0,Y 595.069,Z 482.694,A -85,B 0,C 180,E1 -1186.886,E2 -1186.886} C_VEL
LIN {X 0,Y 595.217,Z 324.564,A -85,B 0,C 180,E1 -1188.851,E2 -1188.851} C_VEL
LIN {X 0,Y 594.731,Z 321.805,A -85,B 0,C 180,E1 -1188.913,E2 -1188.913} C_VEL
LIN {X 0,Y 594.894,Z 296.397,A -85,B 0,C 180,E1 -1191.847,E2 -1191.847} C_VEL
LIN {X 0,Y 595.044,Z 273.243,A -85,B 0,C 180,E1 -1194.572,E2 -1194.572} C_VEL
LIN {X 0,Y 594.966,Z 266.745,A -85,B 0,C 180,E1 -1195.353,E2 -1195.353} C_VEL
LIN {X 0,Y 594.369,Z 264.075,A -85,B 0,C 180,E1 -1195.708,E2 -1195.708} C_VEL
LIN {X 0,Y 594.361,Z 264.078,A -85,B 0,C 180,E1 -1198.227,E2 -1198.227} C_VEL
LIN {X 0,Y 594.372,Z 264.071,A -85,B 0,C 180,E1 -1200.559,E2 -1200.559} C_VEL
LIN {X 0,Y 594.367,Z 264.068,A -85,B 0,C 180,E1 -1202.95,E2 -1202.95} C_VEL
LIN {X 0,Y 594.321,Z 264.074,A -85,B 0,C 180,E1 -1205.41,E2 -1205.41} C_VEL
LIN {X 0,Y 594.368,Z 264.075,A -85,B 0,C 180,E1 -1207.941,E2 -1207.941} C_VEL
LIN {X 0,Y 594.352,Z 264.07,A -85,B 0,C 180,E1 -1210.819,E2 -1210.819} C_VEL
LIN {X 0,Y 594.333,Z 264.072,A -85,B 0,C 180,E1 -1213.301,E2 -1213.301} C_VEL
LIN {X 0,Y 594.334,Z 264.078,A -85,B 0,C 180,E1 -1216.162,E2 -1216.162} C_VEL
LIN {X 0,Y 594.355,Z 264.07,A -85,B 0,C 180,E1 -1218.534,E2 -1218.534} C_VEL
LIN {X 0,Y 594.355,Z 264.07,A -85,B 0,C 180,E1 -1221.297,E2 -1221.297} C_VEL
LIN {X 0,Y 594.333,Z 264.08,A -85,B 0,C 180,E1 -1223.754,E2 -1223.754} C_VEL
LIN {X 0,Y 594.349,Z 264.073,A -85,B 0,C 180,E1 -1226.237,E2 -1226.237} C_VEL
LIN {X 0,Y 594.345,Z 264.07,A -85,B 0,C 180,E1 -1228.648,E2 -1228.648} C_VEL
LIN {X 0,Y 594.362,Z 264.068,A -85,B 0,C 180,E1 -1231.043,E2 -1231.043} C_VEL
LIN {X 0,Y 594.324,Z 264.077,A -85,B 0,C 180,E1 -1234.054,E2 -1234.054} C_VEL
LIN {X 0,Y 594.346,Z 264.071,A -85,B 0,C 180,E1 -1236.294,E2 -1236.294} C_VEL
LIN {X 0,Y 594.384,Z 264.068,A -85,B 0,C 180,E1 -1239.224,E2 -1239.224} C_VEL
LIN {X 0,Y 594.307,Z 264.077,A -85,B 0,C 180,E1 -1242.094,E2 -1242.094} C_VEL
LIN {X 0,Y 594.321,Z 264.074,A -85,B 0,C 180,E1 -1244.218,E2 -1244.218} C_VEL
LIN {X 0,Y 594.325,Z 264.072,A -85,B 0,C 180,E1 -1246.32,E2 -1246.32} C_VEL
LIN {X 0,Y 594.347,Z 264.071,A -85,B 0,C 180,E1 -1249.094,E2 -1249.094} C_VEL
LIN {X 0,Y 594.335,Z 264.076,A -85,B 0,C 180,E1 -1251.842,E2 -1251.842} C_VEL
LIN {X 0,Y 594.326,Z 264.075,A -85,B 0,C 180,E1 -1253.891,E2 -1253.891} C_VEL
LIN {X 0,Y 594.317,Z 264.076,A -85,B 0,C 180,E1 -1255.931,E2 -1255.931} C_VEL
LIN {X 0,Y 594.356,Z 264.07,A -85,B 0,C 180,E1 -1257.967,E2 -1257.967} C_VEL
LIN {X 0,Y 594.373,Z 264.068,A -85,B 0,C 180,E1 -1260,E2 -1260} C_VEL
LIN {X 0,Y 594.363,Z 264.069,A -85,B 0,C 180,E1 -1262.711,E2 -1262.711} C_VEL
LIN {X 0,Y 594.382,Z 264.073,A -85,B 0,C 180,E1 -1265.428,E2 -1265.428} C_VEL
LIN {X 0,Y 594.336,Z 264.071,A -85,B 0,C 180,E1 -1268.158,E2 -1268.158} C_VEL
LIN {X 0,Y 594.361,Z 264.075,A -85,B 0,C 180,E1 -1271.067,E2 -1271.067} C_VEL
LIN {X 0,Y 594.353,Z 264.072,A -85,B 0,C 180,E1 -1273.68,E2 -1273.68} C_VEL
LIN {X 0,Y 594.332,Z 264.077,A -85,B 0,C 180,E1 -1275.29,E2 -1275.29} C_VEL
LIN {X 0,Y 593.66,Z 264.157,A -85,B 0,C 180,E1 -1275.856,E2 -1275.856} C_VEL
LIN {X 0,Y 590.793,Z 264.516,A -85,B 0,C 180,E1 -1276.774,E2 -1276.774} C_VEL
LIN {X 0,Y 588.38,Z 264.817,A -85,B 0,C 180,E1 -1277.512,E2 -1277.512} C_VEL
LIN {X 0,Y 587.357,Z 264.94,A -85,B 0,C 180,E1 -1278.082,E2 -1278.082} C_VEL
LIN {X 0,Y 587.28,Z 264.95,A -85,B 0,C 180,E1 -1278.275,E2 -1278.275} C_VEL
LIN {X 0,Y 587.318,Z 264.953,A -85,B 0,C 180,E1 -1281.038,E2 -1281.038} C_VEL
LIN {X 0,Y 587.281,Z 264.95,A -85,B 0,C 180,E1 -1284.009,E2 -1284.009} C_VEL
LIN {X 0,Y 587.323,Z 264.945,A -85,B 0,C 180,E1 -1286.279,E2 -1286.279} C_VEL
LIN {X 0,Y 587.334,Z 264.951,A -85,B 0,C 180,E1 -1289.133,E2 -1289.133} C_VEL
LIN {X 0,Y 587.336,Z 264.943,A -85,B 0,C 180,E1 -1291.837,E2 -1291.837} C_VEL
LIN {X 0,Y 587.335,Z 264.945,A -85,B 0,C 180,E1 -1294.348,E2 -1294.348} C_VEL
LIN {X 0,Y 587.332,Z 264.944,A -85,B 0,C 180,E1 -1297.609,E2 -1297.609} C_VEL
LIN {X 0,Y 587.3,Z 264.949,A -85,B 0,C 180,E1 -1300.256,E2 -1300.256} C_VEL
LIN {X 0,Y 587.307,Z 264.952,A -85,B 0,C 180,E1 -1303.119,E2 -1303.119} C_VEL
LIN {X 0,Y 587.305,Z 264.948,A -85,B 0,C 180,E1 -1306.049,E2 -1306.049} C_VEL
LIN {X 0,Y 587.329,Z 264.951,A -85,B 0,C 180,E1 -1308.926,E2 -1308.926} C_VEL
LIN {X 0,Y 587.315,Z 264.946,A -85,B 0,C 180,E1 -1311.521,E2 -1311.521} C_VEL
LIN {X 0,Y 587.287,Z 264.951,A -85,B 0,C 180,E1 -1314.101,E2 -1314.101} C_VEL
LIN {X 0,Y 587.323,Z 264.954,A -85,B 0,C 180,E1 -1316.604,E2 -1316.604} C_VEL
LIN {X 0,Y 587.331,Z 264.948,A -85,B 0,C 180,E1 -1319.034,E2 -1319.034} C_VEL
LIN {X 0,Y 587.316,Z 264.947,A -85,B 0,C 180,E1 -1321.403,E2 -1321.403} C_VEL
LIN {X 0,Y 587.337,Z 264.944,A -85,B 0,C 180,E1 -1323.824,E2 -1323.824} C_VEL
LIN {X 0,Y 587.321,Z 264.95,A -85,B 0,C 180,E1 -1325.994,E2 -1325.994} C_VEL
LIN {X 0,Y 587.354,Z 265.104,A -85,B 0,C 180,E1 -1327.124,E2 -1327.124} C_VEL
LIN {X 0,Y 587.856,Z 269.094,A -85,B 0,C 180,E1 -1327.693,E2 -1327.693} C_VEL
LIN {X 0,Y 587.733,Z 287.986,A -85,B 0,C 180,E1 -1330.257,E2 -1330.257} C_VEL
LIN {X 0,Y 587.676,Z 292.846,A -85,B 0,C 180,E1 -1330.909,E2 -1330.909} C_VEL
LIN {X 0,Y 588.556,Z 297.955,A -85,B 0,C 180,E1 -1331.016,E2 -1331.016} C_VEL
LIN {X 0,Y 588.291,Z 458.482,A -85,B 0,C 180,E1 -1333.046,E2 -1333.046} C_VEL
LIN {X 0,Y 588.198,Z 474.495,A -85,B 0,C 180,E1 -1333.403,E2 -1333.403} C_VEL
LIN {X 0,Y 588.082,Z 489.049,A -85,B 0,C 180,E1 -1333.868,E2 -1333.868} C_VEL
LIN {X 0,Y 587.995,Z 503.715,A -85,B 0,C 180,E1 -1334.489,E2 -1334.489} C_VEL
LIN {X 0,Y 587.845,Z 517.016,A -85,B 0,C 180,E1 -1335.194,E2 -1335.194} C_VEL
LIN {X 0,Y 587.734,Z 530.181,A -85,B 0,C 180,E1 -1336.048,E2 -1336.048} C_VEL
LIN {X 0,Y 587.559,Z 542.87,A -85,B 0,C 180,E1 -1337.04,E2 -1337.04} C_VEL
LIN {X 0,Y 587.472,Z 554.071,A -85,B 0,C 180,E1 -1338.091,E2 -1338.091} C_VEL
LIN {X 0,Y 587.382,Z 564.953,A -85,B 0,C 180,E1 -1339.313,E2 -1339.313} C_VEL
LIN {X 0,Y 587.285,Z 573.996,A -85,B 0,C 180,E1 -1340.529,E2 -1340.529} C_VEL
LIN {X 0,Y 587.259,Z 581.489,A -85,B 0,C 180,E1 -1341.743,E2 -1341.743} C_VEL
LIN {X 0,Y 587.207,Z 588.493,A -85,B 0,C 180,E1 -1343.126,E2 -1343.126} C_VEL
LIN {X 0,Y 587.198,Z 594.001,A -85,B 0,C 180,E1 -1344.506,E2 -1344.506} C_VEL
LIN {X 0,Y 587.169,Z 598.173,A -85,B 0,C 180,E1 -1345.882,E2 -1345.882} C_VEL
LIN {X 0,Y 587.127,Z 601.114,A -85,B 0,C 180,E1 -1347.256,E2 -1347.256} C_VEL
LIN {X 0,Y 587.143,Z 602.88,A -85,B 0,C 180,E1 -1348.628,E2 -1348.628} C_VEL
LIN {X 0,Y 587.135,Z 603.496,A -85,B 0,C 180,E1 -1350,E2 -1350} C_VEL
LIN {X 0,Y 587.146,Z 602.943,A -85,B 0,C 180,E1 -1351.372,E2 -1351.372} C_VEL
LIN {X 0,Y 587.129,Z 601.259,A -85,B 0,C 180,E1 -1352.744,E2 -1352.744} C_VEL
LIN {X 0,Y 587.169,Z 598.406,A -85,B 0,C 180,E1 -1354.118,E2 -1354.118} C_VEL
LIN {X 0,Y 587.198,Z 594.324,A -85,B 0,C 180,E1 -1355.494,E2 -1355.494} C_VEL
LIN {X 0,Y 587.207,Z 588.913,A -85,B 0,C 180,E1 -1356.874,E2 -1356.874} C_VEL
LIN {X 0,Y 587.254,Z 582.014,A -85,B 0,C 180,E1 -1358.257,E2 -1358.257} C_VEL
LIN {X 0,Y 587.286,Z 573.411,A -85,B 0,C 180,E1 -1359.644,E2 -1359.644} C_VEL
LIN {X 0,Y 587.367,Z 564.261,A -85,B 0,C 180,E1 -1360.862,E2 -1360.862} C_VEL
LIN {X 0,Y 587.447,Z 554.933,A -85,B 0,C 180,E1 -1361.91,E2 -1361.91} C_VEL
LIN {X 0,Y 587.589,Z 542.893,A -85,B 0,C 180,E1 -1363.047,E2 -1363.047} C_VEL
LIN {X 0,Y 587.709,Z 529.8,A -85,B 0,C 180,E1 -1364.069,E2 -1364.069} C_VEL
LIN {X 0,Y 587.808,Z 517.042,A -85,B 0,C 180,E1 -1364.895,E2 -1364.895} C_VEL
LIN {X 0,Y 587.994,Z 503.741,A -85,B 0,C 180,E1 -1365.6,E2 -1365.6} C_VEL
LIN {X 0,Y 588.082,Z 489.067,A -85,B 0,C 180,E1 -1366.221,E2 -1366.221} C_VEL
LIN {X 0,Y 588.223,Z 473.352,A -85,B 0,C 180,E1 -1366.718,E2 -1366.718} C_VEL
LIN {X 0,Y 588.282,Z 458.457,A -85,B 0,C 180,E1 -1367.045,E2 -1367.045} C_VEL
LIN {X 0,Y 588.551,Z 297.668,A -85,B 0,C 180,E1 -1369.078,E2 -1369.078} C_VEL
LIN {X 0,Y 587.705,Z 292.831,A -85,B 0,C 180,E1 -1369.182,E2 -1369.182} C_VEL
LIN {X 0,Y 587.866,Z 272.451,A -85,B 0,C 180,E1 -1371.937,E2 -1371.937} C_VEL
LIN {X 0,Y 587.772,Z 267.384,A -85,B 0,C 180,E1 -1372.635,E2 -1372.635} C_VEL
LIN {X 0,Y 587.33,Z 264.951,A -85,B 0,C 180,E1 -1373.025,E2 -1373.025} C_VEL
LIN {X 0,Y 587.333,Z 264.954,A -85,B 0,C 180,E1 -1375.516,E2 -1375.516} C_VEL
LIN {X 0,Y 587.343,Z 264.949,A -85,B 0,C 180,E1 -1377.817,E2 -1377.817} C_VEL
LIN {X 0,Y 587.328,Z 264.945,A -85,B 0,C 180,E1 -1380.508,E2 -1380.508} C_VEL
LIN {X 0,Y 587.335,Z 264.948,A -85,B 0,C 180,E1 -1383.111,E2 -1383.111} C_VEL
LIN {X 0,Y 587.34,Z 264.952,A -85,B 0,C 180,E1 -1385.543,E2 -1385.543} C_VEL
LIN {X 0,Y 587.319,Z 264.946,A -85,B 0,C 180,E1 -1388.479,E2 -1388.479} C_VEL
LIN {X 0,Y 587.331,Z 264.95,A -85,B 0,C 180,E1 -1391.156,E2 -1391.156} C_VEL
LIN {X 0,Y 587.305,Z 264.948,A -85,B 0,C 180,E1 -1394.111,E2 -1394.111} C_VEL
LIN {X 0,Y 587.307,Z 264.952,A -85,B 0,C 180,E1 -1396.993,E2 -1396.993} C_VEL
LIN {X 0,Y 587.301,Z 264.95,A -85,B 0,C 180,E1 -1399.744,E2 -1399.744} C_VEL
LIN {X 0,Y 587.333,Z 264.943,A -85,B 0,C 180,E1 -1402.391,E2 -1402.391} C_VEL
LIN {X 0,Y 587.338,Z 264.945,A -85,B 0,C 180,E1 -1405.651,E2 -1405.651} C_VEL
LIN {X 0,Y 587.336,Z 264.942,A -85,B 0,C 180,E1 -1408.231,E2 -1408.231} C_VEL
LIN {X 0,Y 587.335,Z 264.948,A -85,B 0,C 180,E1 -1410.866,E2 -1410.866} C_VEL
LIN {X 0,Y 587.324,Z 264.945,A -85,B 0,C 180,E1 -1413.721,E2 -1413.721} C_VEL
LIN {X 0,Y 587.291,Z 264.949,A -85,B 0,C 180,E1 -1415.991,E2 -1415.991} C_VEL
LIN {X 0,Y 587.318,Z 264.955,A -85,B 0,C 180,E1 -1418.962,E2 -1418.962} C_VEL
LIN {X 0,Y 587.328,Z 264.95,A -85,B 0,C 180,E1 -1421.15,E2 -1421.15} C_VEL
LIN {X 0,Y 587.3,Z 264.948,A -85,B 0,C 180,E1 -1424.024,E2 -1424.024} C_VEL
LIN {X 0,Y 587.295,Z 264.958,A -85,B 0,C 180,E1 -1426.858,E2 -1426.858} C_VEL
LIN {X 0,Y 587.322,Z 264.953,A -85,B 0,C 180,E1 -1428.962,E2 -1428.962} C_VEL
LIN {X 0,Y 587.303,Z 264.947,A -85,B 0,C 180,E1 -1431.744,E2 -1431.744} C_VEL
LIN {X 0,Y 587.346,Z 264.948,A -85,B 0,C 180,E1 -1434.507,E2 -1434.507} C_VEL
LIN {X 0,Y 587.337,Z 264.945,A -85,B 0,C 180,E1 -1437.256,E2 -1437.256} C_VEL
LIN {X 0,Y 587.346,Z 264.942,A -85,B 0,C 180,E1 -1440,E2 -1440} C_VEL
LIN {X 0,Y 587.36,Z 264.948,A -85,B 0,C 180,E1 -1442.743,E2 -1442.743} C_VEL
LIN {X 0,Y 587.309,Z 264.946,A -85,B 0,C 180,E1 -1445.493,E2 -1445.493} C_VEL
LIN {X 0,Y 587.288,Z 264.949,A -85,B 0,C 180,E1 -1447.564,E2 -1447.564} C_VEL
LIN {X 0,Y 587.285,Z 264.956,A -85,B 0,C 180,E1 -1450.341,E2 -1450.341} C_VEL
LIN {X 0,Y 587.279,Z 264.951,A -85,B 0,C 180,E1 -1453.142,E2 -1453.142} C_VEL
LIN {X 0,Y 587.297,Z 264.948,A -85,B 0,C 180,E1 -1455.264,E2 -1455.264} C_VEL
LIN {X 0,Y 587.263,Z 264.952,A -85,B 0,C 180,E1 -1457.409,E2 -1457.409} C_VEL
LIN {X 0,Y 587.282,Z 264.95,A -85,B 0,C 180,E1 -1459.577,E2 -1459.577} C_VEL
LIN {X 0,Y 587.292,Z 264.95,A -85,B 0,C 180,E1 -1461.775,E2 -1461.775} C_VEL
LIN {X 0,Y 587.292,Z 264.952,A -85,B 0,C 180,E1 -1464.761,E2 -1464.761} C_VEL
LIN {X 0,Y 587.286,Z 264.951,A -85,B 0,C 180,E1 -1467.684,E2 -1467.684} C_VEL
LIN {X 0,Y 587.301,Z 264.957,A -85,B 0,C 180,E1 -1470.172,E2 -1470.172} C_VEL
LIN {X 0,Y 587.324,Z 264.948,A -85,B 0,C 180,E1 -1472.58,E2 -1472.58} C_VEL
LIN {X 0,Y 587.283,Z 264.95,A -85,B 0,C 180,E1 -1475.059,E2 -1475.059} C_VEL
LIN {X 0,Y 587.307,Z 264.952,A -85,B 0,C 180,E1 -1477.836,E2 -1477.836} C_VEL
LIN {X 0,Y 587.294,Z 264.954,A -85,B 0,C 180,E1 -1480.256,E2 -1480.256} C_VEL
LIN {X 0,Y 587.291,Z 264.949,A -85,B 0,C 180,E1 -1483.008,E2 -1483.008} C_VEL
LIN {X 0,Y 587.292,Z 264.958,A -85,B 0,C 180,E1 -1486.048,E2 -1486.048} C_VEL
LIN {X 0,Y 587.301,Z 264.947,A -85,B 0,C 180,E1 -1488.929,E2 -1488.929} C_VEL
LIN {X 0,Y 587.308,Z 264.95,A -85,B 0,C 180,E1 -1491.52,E2 -1491.52} C_VEL
LIN {X 0,Y 587.28,Z 264.957,A -85,B 0,C 180,E1 -1494.1,E2 -1494.1} C_VEL
LIN {X 0,Y 587.324,Z 264.946,A -85,B 0,C 180,E1 -1496.604,E2 -1496.604} C_VEL
LIN {X 0,Y 587.328,Z 264.949,A -85,B 0,C 180,E1 -1499.492,E2 -1499.492} C_VEL
LIN {X 0,Y 587.298,Z 264.954,A -85,B 0,C 180,E1 -1502.181,E2 -1502.181} C_VEL
LIN {X 0,Y 587.335,Z 264.977,A -85,B 0,C 180,E1 -1504.078,E2 -1504.078} C_VEL
LIN {X 0,Y 588.24,Z 270.023,A -85,B 0,C 180,E1 -1504.735,E2 -1504.735} C_VEL
LIN {X 0,Y 588.052,Z 293.276,A -85,B 0,C 180,E1 -1507.516,E2 -1507.516} C_VEL
LIN {X 0,Y 587.845,Z 318.245,A -85,B 0,C 180,E1 -1510.443,E2 -1510.443} C_VEL
LIN {X 0,Y 587.814,Z 322.06,A -85,B 0,C 180,E1 -1510.871,E2 -1510.871} C_VEL
LIN {X 0,Y 588.593,Z 326.589,A -85,B 0,C 180,E1 -1510.955,E2 -1510.955} C_VEL
LIN {X 0,Y 588.292,Z 488.517,A -85,B 0,C 180,E1 -1513.002,E2 -1513.002} C_VEL
LIN {X 0,Y 588.216,Z 504.499,A -85,B 0,C 180,E1 -1513.359,E2 -1513.359} C_VEL
LIN {X 0,Y 588.071,Z 519.056,A -85,B 0,C 180,E1 -1513.823,E2 -1513.823} C_VEL
LIN {X 0,Y 587.988,Z 532.775,A -85,B 0,C 180,E1 -1514.4,E2 -1514.4} C_VEL
LIN {X 0,Y 587.836,Z 546.246,A -85,B 0,C 180,E1 -1515.105,E2 -1515.105} C_VEL
LIN {X 0,Y 587.74,Z 559.12,A -85,B 0,C 180,E1 -1515.93,E2 -1515.93} C_VEL
LIN {X 0,Y 587.583,Z 571.292,A -85,B 0,C 180,E1 -1516.865,E2 -1516.865} C_VEL
LIN {X 0,Y 587.453,Z 582.752,A -85,B 0,C 180,E1 -1517.915,E2 -1517.915} C_VEL
LIN {X 0,Y 587.349,Z 592.393,A -85,B 0,C 180,E1 -1518.963,E2 -1518.963} C_VEL
LIN {X 0,Y 587.304,Z 601.858,A -85,B 0,C 180,E1 -1520.182,E2 -1520.182} C_VEL
LIN {X 0,Y 587.264,Z 609.733,A -85,B 0,C 180,E1 -1521.397,E2 -1521.397} C_VEL
LIN {X 0,Y 587.215,Z 617.089,A -85,B 0,C 180,E1 -1522.781,E2 -1522.781} C_VEL
LIN {X 0,Y 587.224,Z 622.924,A -85,B 0,C 180,E1 -1524.161,E2 -1524.161} C_VEL
LIN {X 0,Y 587.136,Z 626.385,A -85,B 0,C 180,E1 -1525.194,E2 -1525.194} C_VEL
LIN {X 0,Y 587.179,Z 629.888,A -85,B 0,C 180,E1 -1526.569,E2 -1526.569} C_VEL
LIN {X 0,Y 587.138,Z 632.193,A -85,B 0,C 180,E1 -1527.942,E2 -1527.942} C_VEL
LIN {X 0,Y 587.137,Z 633.35,A -85,B 0,C 180,E1 -1529.314,E2 -1529.314} C_VEL
LIN {X 0,Y 587.137,Z 633.349,A -85,B 0,C 180,E1 -1530.686,E2 -1530.686} C_VEL
LIN {X 0,Y 587.138,Z 632.193,A -85,B 0,C 180,E1 -1532.058,E2 -1532.058} C_VEL
LIN {X 0,Y 587.179,Z 629.887,A -85,B 0,C 180,E1 -1533.431,E2 -1533.431} C_VEL
LIN {X 0,Y 587.136,Z 626.385,A -85,B 0,C 180,E1 -1534.806,E2 -1534.806} C_VEL
LIN {X 0,Y 587.178,Z 621.609,A -85,B 0,C 180,E1 -1536.184,E2 -1536.184} C_VEL
LIN {X 0,Y 587.23,Z 615.425,A -85,B 0,C 180,E1 -1537.565,E2 -1537.565} C_VEL
LIN {X 0,Y 587.266,Z 607.652,A -85,B 0,C 180,E1 -1538.95,E2 -1538.95} C_VEL
LIN {X 0,Y 587.351,Z 599.372,A -85,B 0,C 180,E1 -1540.165,E2 -1540.165} C_VEL
LIN {X 0,Y 587.399,Z 589.398,A -85,B 0,C 180,E1 -1541.385,E2 -1541.385} C_VEL
LIN {X 0,Y 587.521,Z 579.194,A -85,B 0,C 180,E1 -1542.434,E2 -1542.434} C_VEL
LIN {X 0,Y 587.629,Z 567.023,A -85,B 0,C 180,E1 -1543.486,E2 -1543.486} C_VEL
LIN {X 0,Y 587.773,Z 554.063,A -85,B 0,C 180,E1 -1544.416,E2 -1544.416} C_VEL
LIN {X 0,Y 587.887,Z 539.875,A -85,B 0,C 180,E1 -1545.248,E2 -1545.248} C_VEL
LIN {X 0,Y 588.051,Z 525.807,A -85,B 0,C 180,E1 -1545.91,E2 -1545.91} C_VEL
LIN {X 0,Y 588.17,Z 511.318,A -85,B 0,C 180,E1 -1546.441,E2 -1546.441} C_VEL
LIN {X 0,Y 588.28,Z 496.28,A -85,B 0,C 180,E1 -1546.844,E2 -1546.844} C_VEL
LIN {X 0,Y 588.321,Z 481.087,A -85,B 0,C 180,E1 -1547.11,E2 -1547.11} C_VEL
LIN {X 0,Y 588.504,Z 325.448,A -85,B 0,C 180,E1 -1549.063,E2 -1549.063} C_VEL
LIN {X 0,Y 587.804,Z 321.776,A -85,B 0,C 180,E1 -1549.148,E2 -1549.148} C_VEL
LIN {X 0,Y 588.032,Z 296.397,A -85,B 0,C 180,E1 -1552.115,E2 -1552.115} C_VEL
LIN {X 0,Y 588.232,Z 273.145,A -85,B 0,C 180,E1 -1554.888,E2 -1554.888} C_VEL
LIN {X 0,Y 588.102,Z 268.306,A -85,B 0,C 180,E1 -1555.48,E2 -1555.48} C_VEL
LIN {X 0,Y 587.329,Z 264.953,A -85,B 0,C 180,E1 -1555.947,E2 -1555.947} C_VEL
LIN {X 0,Y 587.34,Z 264.944,A -85,B 0,C 180,E1 -1559.132,E2 -1559.132} C_VEL
LIN {X 0,Y 587.334,Z 264.949,A -85,B 0,C 180,E1 -1561.834,E2 -1561.834} C_VEL
LIN {X 0,Y 587.332,Z 264.95,A -85,B 0,C 180,E1 -1564.345,E2 -1564.345} C_VEL
LIN {X 0,Y 587.314,Z 264.949,A -85,B 0,C 180,E1 -1567.609,E2 -1567.609} C_VEL
LIN {X 0,Y 587.298,Z 264.955,A -85,B 0,C 180,E1 -1570.254,E2 -1570.254} C_VEL
LIN {X 0,Y 587.278,Z 264.951,A -85,B 0,C 180,E1 -1573.114,E2 -1573.114} C_VEL
LIN {X 0,Y 587.29,Z 264.958,A -85,B 0,C 180,E1 -1576.046,E2 -1576.046} C_VEL
LIN {X 0,Y 587.298,Z 264.948,A -85,B 0,C 180,E1 -1578.84,E2 -1578.84} C_VEL
LIN {X 0,Y 587.304,Z 264.951,A -85,B 0,C 180,E1 -1581.519,E2 -1581.519} C_VEL
LIN {X 0,Y 587.265,Z 264.958,A -85,B 0,C 180,E1 -1584.098,E2 -1584.098} C_VEL
LIN {X 0,Y 587.323,Z 264.944,A -85,B 0,C 180,E1 -1586.888,E2 -1586.888} C_VEL
LIN {X 0,Y 587.309,Z 264.952,A -85,B 0,C 180,E1 -1589.492,E2 -1589.492} C_VEL
LIN {X 0,Y 587.289,Z 264.952,A -85,B 0,C 180,E1 -1592.179,E2 -1592.179} C_VEL
LIN {X 0,Y 587.279,Z 264.951,A -85,B 0,C 180,E1 -1594.481,E2 -1594.481} C_VEL
LIN {X 0,Y 587.292,Z 264.95,A -85,B 0,C 180,E1 -1597.134,E2 -1597.134} C_VEL
LIN {X 0,Y 587.303,Z 264.955,A -85,B 0,C 180,E1 -1599.694,E2 -1599.694} C_VEL
LIN {X 0,Y 587.264,Z 264.957,A -85,B 0,C 180,E1 -1601.871,E2 -1601.871} C_VEL
LIN {X 0,Y 587.283,Z 264.953,A -85,B 0,C 180,E1 -1604.024,E2 -1604.024} C_VEL
LIN {X 0,Y 587.309,Z 264.947,A -85,B 0,C 180,E1 -1606.153,E2 -1606.153} C_VEL
LIN {X 0,Y 587.274,Z 264.95,A -85,B 0,C 180,E1 -1608.961,E2 -1608.961} C_VEL
LIN {X 0,Y 587.302,Z 264.953,A -85,B 0,C 180,E1 -1611.744,E2 -1611.744} C_VEL
LIN {X 0,Y 587.285,Z 264.953,A -85,B 0,C 180,E1 -1613.817,E2 -1613.817} C_VEL
LIN {X 0,Y 587.274,Z 264.954,A -85,B 0,C 180,E1 -1615.883,E2 -1615.883} C_VEL
LIN {X 0,Y 587.329,Z 264.945,A -85,B 0,C 180,E1 -1617.943,E2 -1617.943} C_VEL
LIN {X 0,Y 587.344,Z 264.944,A -85,B 0,C 180,E1 -1620,E2 -1620} C_VEL
LIN {X 0,Y 587.333,Z 264.945,A -85,B 0,C 180,E1 -1622.744,E2 -1622.744} C_VEL
LIN {X 0,Y 587.343,Z 264.949,A -85,B 0,C 180,E1 -1625.493,E2 -1625.493} C_VEL
LIN {X 0,Y 587.303,Z 264.947,A -85,B 0,C 180,E1 -1628.256,E2 -1628.256} C_VEL
LIN {X 0,Y 587.334,Z 264.952,A -85,B 0,C 180,E1 -1631.134,E2 -1631.134} C_VEL
LIN {X 0,Y 587.295,Z 264.948,A -85,B 0,C 180,E1 -1634.239,E2 -1634.239} C_VEL
LIN {X 0,Y 587.316,Z 264.95,A -85,B 0,C 180,E1 -1636.808,E2 -1636.808} C_VEL
LIN {X 0,Y 587.28,Z 264.95,A -85,B 0,C 180,E1 -1638.275,E2 -1638.275} C_VEL
LIN {X 0,Y 586.643,Z 265.036,A -85,B 0,C 180,E1 -1638.847,E2 -1638.847} C_VEL
LIN {X 0,Y 583.836,Z 265.389,A -85,B 0,C 180,E1 -1639.776,E2 -1639.776} C_VEL
LIN {X 0,Y 581.432,Z 265.691,A -85,B 0,C 180,E1 -1640.523,E2 -1640.523} C_VEL
LIN {X 0,Y 580.372,Z 265.819,A -85,B 0,C 180,E1 -1641.1,E2 -1641.1} C_VEL
LIN {X 0,Y 580.271,Z 265.829,A -85,B 0,C 180,E1 -1641.295,E2 -1641.295} C_VEL
LIN {X 0,Y 580.241,Z 265.83,A -85,B 0,C 180,E1 -1643.56,E2 -1643.56} C_VEL
LIN {X 0,Y 580.276,Z 265.823,A -85,B 0,C 180,E1 -1646.334,E2 -1646.334} C_VEL
LIN {X 0,Y 580.283,Z 265.827,A -85,B 0,C 180,E1 -1649.309,E2 -1649.309} C_VEL
LIN {X 0,Y 580.286,Z 265.821,A -85,B 0,C 180,E1 -1652.201,E2 -1652.201} C_VEL
LIN {X 0,Y 580.281,Z 265.828,A -85,B 0,C 180,E1 -1654.697,E2 -1654.697} C_VEL
LIN {X 0,Y 580.288,Z 265.825,A -85,B 0,C 180,E1 -1657.269,E2 -1657.269} C_VEL
LIN {X 0,Y 580.279,Z 265.824,A -85,B 0,C 180,E1 -1660.271,E2 -1660.271} C_VEL
LIN {X 0,Y 580.269,Z 265.832,A -85,B 0,C 180,E1 -1662.707,E2 -1662.707} C_VEL
LIN {X 0,Y 580.248,Z 265.827,A -85,B 0,C 180,E1 -1665.612,E2 -1665.612} C_VEL
LIN {X 0,Y 580.269,Z 265.826,A -85,B 0,C 180,E1 -1668.232,E2 -1668.232} C_VEL
LIN {X 0,Y 580.268,Z 265.829,A -85,B 0,C 180,E1 -1670.966,E2 -1670.966} C_VEL
LIN {X 0,Y 580.263,Z 265.824,A -85,B 0,C 180,E1 -1673.597,E2 -1673.597} C_VEL
LIN {X 0,Y 580.298,Z 265.823,A -85,B 0,C 180,E1 -1676.145,E2 -1676.145} C_VEL
LIN {X 0,Y 580.28,Z 265.832,A -85,B 0,C 180,E1 -1678.616,E2 -1678.616} C_VEL
LIN {X 0,Y 580.287,Z 265.825,A -85,B 0,C 180,E1 -1681.024,E2 -1681.024} C_VEL
LIN {X 0,Y 580.288,Z 265.822,A -85,B 0,C 180,E1 -1683.667,E2 -1683.667} C_VEL
LIN {X 0,Y 580.293,Z 265.823,A -85,B 0,C 180,E1 -1685.684,E2 -1685.684} C_VEL
LIN {X 0,Y 580.308,Z 265.966,A -85,B 0,C 180,E1 -1686.95,E2 -1686.95} C_VEL
LIN {X 0,Y 580.956,Z 270.448,A -85,B 0,C 180,E1 -1687.601,E2 -1687.601} C_VEL
LIN {X 0,Y 580.785,Z 289.339,A -85,B 0,C 180,E1 -1690.195,E2 -1690.195} C_VEL
LIN {X 0,Y 580.75,Z 292.929,A -85,B 0,C 180,E1 -1690.683,E2 -1690.683} C_VEL
LIN {X 0,Y 581.841,Z 298.687,A -85,B 0,C 180,E1 -1690.797,E2 -1690.797} C_VEL
LIN {X 0,Y 581.515,Z 458.319,A -85,B 0,C 180,E1 -1692.839,E2 -1692.839} C_VEL
LIN {X 0,Y 581.41,Z 473.742,A -85,B 0,C 180,E1 -1693.181,E2 -1693.181} C_VEL
LIN {X 0,Y 581.233,Z 489.063,A -85,B 0,C 180,E1 -1693.673,E2 -1693.673} C_VEL
LIN {X 0,Y 581.117,Z 503.724,A -85,B 0,C 180,E1 -1694.3,E2 -1694.3} C_VEL
LIN {X 0,Y 580.925,Z 517.029,A -85,B 0,C 180,E1 -1695.014,E2 -1695.014} C_VEL
LIN {X 0,Y 580.791,Z 530.377,A -85,B 0,C 180,E1 -1695.89,E2 -1695.89} C_VEL
LIN {X 0,Y 580.593,Z 542.878,A -85,B 0,C 180,E1 -1696.882,E2 -1696.882} C_VEL
LIN {X 0,Y 580.47,Z 554.077,A -85,B 0,C 180,E1 -1697.945,E2 -1697.945} C_VEL
LIN {X 0,Y 580.337,Z 565.114,A -85,B 0,C 180,E1 -1699.201,E2 -1699.201} C_VEL
LIN {X 0,Y 580.239,Z 573.999,A -85,B 0,C 180,E1 -1700.413,E2 -1700.413} C_VEL
LIN {X 0,Y 580.196,Z 581.492,A -85,B 0,C 180,E1 -1701.642,E2 -1701.642} C_VEL
LIN {X 0,Y 580.139,Z 588.496,A -85,B 0,C 180,E1 -1703.042,E2 -1703.042} C_VEL
LIN {X 0,Y 580.127,Z 594.004,A -85,B 0,C 180,E1 -1704.439,E2 -1704.439} C_VEL
LIN {X 0,Y 580.088,Z 598.174,A -85,B 0,C 180,E1 -1705.831,E2 -1705.831} C_VEL
LIN {X 0,Y 580.038,Z 601.114,A -85,B 0,C 180,E1 -1707.222,E2 -1707.222} C_VEL
LIN {X 0,Y 580.043,Z 602.88,A -85,B 0,C 180,E1 -1708.611,E2 -1708.611} C_VEL
LIN {X 0,Y 580.035,Z 603.496,A -85,B 0,C 180,E1 -1710,E2 -1710} C_VEL
LIN {X 0,Y 580.045,Z 602.943,A -85,B 0,C 180,E1 -1711.389,E2 -1711.389} C_VEL
LIN {X 0,Y 580.04,Z 601.259,A -85,B 0,C 180,E1 -1712.778,E2 -1712.778} C_VEL
LIN {X 0,Y 580.088,Z 598.405,A -85,B 0,C 180,E1 -1714.169,E2 -1714.169} C_VEL
LIN {X 0,Y 580.123,Z 594.322,A -85,B 0,C 180,E1 -1715.562,E2 -1715.562} C_VEL
LIN {X 0,Y 580.139,Z 588.91,A -85,B 0,C 180,E1 -1716.958,E2 -1716.958} C_VEL
LIN {X 0,Y 580.19,Z 582.011,A -85,B 0,C 180,E1 -1718.358,E2 -1718.358} C_VEL
LIN {X 0,Y 580.235,Z 573.406,A -85,B 0,C 180,E1 -1719.763,E2 -1719.763} C_VEL
LIN {X 0,Y 580.308,Z 563.831,A -85,B 0,C 180,E1 -1721.047,E2 -1721.047} C_VEL
LIN {X 0,Y 580.472,Z 553.203,A -85,B 0,C 180,E1 -1722.232,E2 -1722.232} C_VEL
LIN {X 0,Y 580.606,Z 541.829,A -85,B 0,C 180,E1 -1723.296,E2 -1723.296} C_VEL
LIN {X 0,Y 580.759,Z 529.076,A -85,B 0,C 180,E1 -1724.291,E2 -1724.291} C_VEL
LIN {X 0,Y 580.924,Z 515.469,A -85,B 0,C 180,E1 -1725.166,E2 -1725.166} C_VEL
LIN {X 0,Y 581.122,Z 501.794,A -85,B 0,C 180,E1 -1725.88,E2 -1725.88} C_VEL
LIN {X 0,Y 581.266,Z 487.805,A -85,B 0,C 180,E1 -1726.462,E2 -1726.462} C_VEL
LIN {X 0,Y 581.443,Z 472.798,A -85,B 0,C 180,E1 -1726.932,E2 -1726.932} C_VEL
LIN {X 0,Y 581.497,Z 458.499,A -85,B 0,C 180,E1 -1727.248,E2 -1727.248} C_VEL
LIN {X 0,Y 581.795,Z 298.099,A -85,B 0,C 180,E1 -1729.302,E2 -1729.302} C_VEL
LIN {X 0,Y 580.78,Z 292.913,A -85,B 0,C 180,E1 -1729.408,E2 -1729.408} C_VEL
LIN {X 0,Y 580.974,Z 272.446,A -85,B 0,C 180,E1 -1732.211,E2 -1732.211} C_VEL
LIN {X 0,Y 580.801,Z 268.396,A -85,B 0,C 180,E1 -1732.781,E2 -1732.781} C_VEL
LIN {X 0,Y 580.285,Z 265.83,A -85,B 0,C 180,E1 -1733.166,E2 -1733.166} C_VEL
LIN {X 0,Y 580.291,Z 265.827,A -85,B 0,C 180,E1 -1735.848,E2 -1735.848} C_VEL
LIN {X 0,Y 580.295,Z 265.823,A -85,B 0,C 180,E1 -1738.185,E2 -1738.185} C_VEL
LIN {X 0,Y 580.282,Z 265.823,A -85,B 0,C 180,E1 -1740.694,E2 -1740.694} C_VEL
LIN {X 0,Y 580.3,Z 265.828,A -85,B 0,C 180,E1 -1743.315,E2 -1743.315} C_VEL
LIN {X 0,Y 580.266,Z 265.83,A -85,B 0,C 180,E1 -1745.759,E2 -1745.759} C_VEL
LIN {X 0,Y 580.28,Z 265.824,A -85,B 0,C 180,E1 -1748.146,E2 -1748.146} C_VEL
LIN {X 0,Y 580.293,Z 265.822,A -85,B 0,C 180,E1 -1750.842,E2 -1750.842} C_VEL
LIN {X 0,Y 580.266,Z 265.829,A -85,B 0,C 180,E1 -1753.658,E2 -1753.658} C_VEL
LIN {X 0,Y 580.267,Z 265.825,A -85,B 0,C 180,E1 -1756.609,E2 -1756.609} C_VEL
LIN {X 0,Y 580.289,Z 265.828,A -85,B 0,C 180,E1 -1759.156,E2 -1759.156} C_VEL
LIN {X 0,Y 580.277,Z 265.822,A -85,B 0,C 180,E1 -1761.927,E2 -1761.927} C_VEL
LIN {X 0,Y 580.246,Z 265.826,A -85,B 0,C 180,E1 -1764.452,E2 -1764.452} C_VEL
LIN {X 0,Y 580.277,Z 265.83,A -85,B 0,C 180,E1 -1766.974,E2 -1766.974} C_VEL
LIN {X 0,Y 580.279,Z 265.825,A -85,B 0,C 180,E1 -1769.424,E2 -1769.424} C_VEL
LIN {X 0,Y 580.284,Z 265.822,A -85,B 0,C 180,E1 -1772.141,E2 -1772.141} C_VEL
LIN {X 0,Y 580.275,Z 265.831,A -85,B 0,C 180,E1 -1774.919,E2 -1774.919} C_VEL
LIN {X 0,Y 580.243,Z 265.826,A -85,B 0,C 180,E1 -1777.946,E2 -1777.946} C_VEL
LIN {X 0,Y 580.281,Z 265.832,A -85,B 0,C 180,E1 -1780.913,E2 -1780.913} C_VEL
LIN {X 0,Y 580.252,Z 265.826,A -85,B 0,C 180,E1 -1783.825,E2 -1783.825} C_VEL
LIN {X 0,Y 580.252,Z 265.833,A -85,B 0,C 180,E1 -1786.695,E2 -1786.695} C_VEL
LIN {X 0,Y 580.291,Z 265.831,A -85,B 0,C 180,E1 -1788.827,E2 -1788.827} C_VEL
LIN {X 0,Y 580.277,Z 265.822,A -85,B 0,C 180,E1 -1791.643,E2 -1791.643} C_VEL
LIN {X 0,Y 580.308,Z 265.824,A -85,B 0,C 180,E1 -1794.44,E2 -1794.44} C_VEL
LIN {X 0,Y 580.306,Z 265.821,A -85,B 0,C 180,E1 -1797.223,E2 -1797.223} C_VEL
LIN {X 0,Y 580.318,Z 265.818,A -85,B 0,C 180,E1 -1800,E2 -1800} C_VEL
LIN {X 0,Y 580.323,Z 265.824,A -85,B 0,C 180,E1 -1802.777,E2 -1802.777} C_VEL
LIN {X 0,Y 580.277,Z 265.822,A -85,B 0,C 180,E1 -1805.56,E2 -1805.56} C_VEL
LIN {X 0,Y 580.24,Z 265.827,A -85,B 0,C 180,E1 -1807.656,E2 -1807.656} C_VEL
LIN {X 0,Y 580.253,Z 265.834,A -85,B 0,C 180,E1 -1810.468,E2 -1810.468} C_VEL
LIN {X 0,Y 580.274,Z 265.83,A -85,B 0,C 180,E1 -1812.592,E2 -1812.592} C_VEL
LIN {X 0,Y 580.265,Z 265.83,A -85,B 0,C 180,E1 -1814.735,E2 -1814.735} C_VEL
LIN {X 0,Y 580.228,Z 265.829,A -85,B 0,C 180,E1 -1817.626,E2 -1817.626} C_VEL
LIN {X 0,Y 580.261,Z 265.827,A -85,B 0,C 180,E1 -1819.824,E2 -1819.824} C_VEL
LIN {X 0,Y 580.245,Z 265.831,A -85,B 0,C 180,E1 -1822.054,E2 -1822.054} C_VEL
LIN {X 0,Y 580.25,Z 265.829,A -85,B 0,C 180,E1 -1824.718,E2 -1824.718} C_VEL
LIN {X 0,Y 580.23,Z 265.829,A -85,B 0,C 180,E1 -1827.405,E2 -1827.405} C_VEL
LIN {X 0,Y 580.251,Z 265.829,A -85,B 0,C 180,E1 -1829.775,E2 -1829.775} C_VEL
LIN {X 0,Y 580.284,Z 265.832,A -85,B 0,C 180,E1 -1832.201,E2 -1832.201} C_VEL
LIN {X 0,Y 580.26,Z 265.827,A -85,B 0,C 180,E1 -1834.698,E2 -1834.698} C_VEL
LIN {X 0,Y 580.256,Z 265.825,A -85,B 0,C 180,E1 -1837.272,E2 -1837.272} C_VEL
LIN {X 0,Y 580.274,Z 265.828,A -85,B 0,C 180,E1 -1840.27,E2 -1840.27} C_VEL
LIN {X 0,Y 580.26,Z 265.826,A -85,B 0,C 180,E1 -1842.708,E2 -1842.708} C_VEL
LIN {X 0,Y 580.242,Z 265.831,A -85,B 0,C 180,E1 -1845.612,E2 -1845.612} C_VEL
LIN {X 0,Y 580.241,Z 265.833,A -85,B 0,C 180,E1 -1848.229,E2 -1848.229} C_VEL
LIN {X 0,Y 580.26,Z 265.825,A -85,B 0,C 180,E1 -1850.965,E2 -1850.965} C_VEL
LIN {X 0,Y 580.239,Z 265.832,A -85,B 0,C 180,E1 -1853.595,E2 -1853.595} C_VEL
LIN {X 0,Y 580.304,Z 265.826,A -85,B 0,C 180,E1 -1856.146,E2 -1856.146} C_VEL
LIN {X 0,Y 580.265,Z 265.825,A -85,B 0,C 180,E1 -1858.615,E2 -1858.615} C_VEL
LIN {X 0,Y 580.282,Z 265.824,A -85,B 0,C 180,E1 -1861.024,E2 -1861.024} C_VEL
LIN {X 0,Y 580.281,Z 265.859,A -85,B 0,C 180,E1 -1863.855,E2 -1863.855} C_VEL
LIN {X 0,Y 581.411,Z 271.427,A -85,B 0,C 180,E1 -1864.589,E2 -1864.589} C_VEL
LIN {X 0,Y 581.243,Z 291.889,A -85,B 0,C 180,E1 -1867.071,E2 -1867.071} C_VEL
LIN {X 0,Y 580.967,Z 316.685,A -85,B 0,C 180,E1 -1870.018,E2 -1870.018} C_VEL
LIN {X 0,Y 580.896,Z 321.909,A -85,B 0,C 180,E1 -1870.631,E2 -1870.631} C_VEL
LIN {X 0,Y 581.899,Z 327.773,A -85,B 0,C 180,E1 -1870.742,E2 -1870.742} C_VEL
LIN {X 0,Y 581.517,Z 488.074,A -85,B 0,C 180,E1 -1872.79,E2 -1872.79} C_VEL
LIN {X 0,Y 581.431,Z 503.724,A -85,B 0,C 180,E1 -1873.137,E2 -1873.137} C_VEL
LIN {X 0,Y 581.243,Z 519.054,A -85,B 0,C 180,E1 -1873.628,E2 -1873.628} C_VEL
LIN {X 0,Y 581.124,Z 532.778,A -85,B 0,C 180,E1 -1874.211,E2 -1874.211} C_VEL
LIN {X 0,Y 580.943,Z 546.249,A -85,B 0,C 180,E1 -1874.925,E2 -1874.925} C_VEL
LIN {X 0,Y 580.804,Z 559.485,A -85,B 0,C 180,E1 -1875.784,E2 -1875.784} C_VEL
LIN {X 0,Y 580.608,Z 571.293,A -85,B 0,C 180,E1 -1876.704,E2 -1876.704} C_VEL
LIN {X 0,Y 580.478,Z 582.752,A -85,B 0,C 180,E1 -1877.768,E2 -1877.768} C_VEL
LIN {X 0,Y 580.308,Z 593.452,A -85,B 0,C 180,E1 -1878.953,E2 -1878.953} C_VEL
LIN {X 0,Y 580.268,Z 601.859,A -85,B 0,C 180,E1 -1880.062,E2 -1880.062} C_VEL
LIN {X 0,Y 580.214,Z 609.734,A -85,B 0,C 180,E1 -1881.292,E2 -1881.292} C_VEL
LIN {X 0,Y 580.13,Z 617.09,A -85,B 0,C 180,E1 -1882.692,E2 -1882.692} C_VEL
LIN {X 0,Y 580.129,Z 622.924,A -85,B 0,C 180,E1 -1884.09,E2 -1884.09} C_VEL
LIN {X 0,Y 580.041,Z 626.385,A -85,B 0,C 180,E1 -1885.135,E2 -1885.135} C_VEL
LIN {X 0,Y 580.104,Z 629.889,A -85,B 0,C 180,E1 -1886.527,E2 -1886.527} C_VEL
LIN {X 0,Y 580.037,Z 632.193,A -85,B 0,C 180,E1 -1887.917,E2 -1887.917} C_VEL
LIN {X 0,Y 580.038,Z 633.349,A -85,B 0,C 180,E1 -1889.306,E2 -1889.306} C_VEL
LIN {X 0,Y 580.038,Z 633.349,A -85,B 0,C 180,E1 -1890.694,E2 -1890.694} C_VEL
LIN {X 0,Y 580.037,Z 632.192,A -85,B 0,C 180,E1 -1892.083,E2 -1892.083} C_VEL
LIN {X 0,Y 580.104,Z 629.887,A -85,B 0,C 180,E1 -1893.473,E2 -1893.473} C_VEL
LIN {X 0,Y 580.041,Z 626.385,A -85,B 0,C 180,E1 -1894.865,E2 -1894.865} C_VEL
LIN {X 0,Y 580.091,Z 621.609,A -85,B 0,C 180,E1 -1896.26,E2 -1896.26} C_VEL
LIN {X 0,Y 580.165,Z 615.425,A -85,B 0,C 180,E1 -1897.657,E2 -1897.657} C_VEL
LIN {X 0,Y 580.207,Z 607.651,A -85,B 0,C 180,E1 -1899.06,E2 -1899.06} C_VEL
LIN {X 0,Y 580.308,Z 599.371,A -85,B 0,C 180,E1 -1900.29,E2 -1900.29} C_VEL
LIN {X 0,Y 580.382,Z 589.398,A -85,B 0,C 180,E1 -1901.525,E2 -1901.525} C_VEL
LIN {X 0,Y 580.541,Z 579.193,A -85,B 0,C 180,E1 -1902.586,E2 -1902.586} C_VEL
LIN {X 0,Y 580.677,Z 567.024,A -85,B 0,C 180,E1 -1903.651,E2 -1903.651} C_VEL
LIN {X 0,Y 580.874,Z 553.533,A -85,B 0,C 180,E1 -1904.625,E2 -1904.625} C_VEL
LIN {X 0,Y 581.018,Z 539.877,A -85,B 0,C 180,E1 -1905.433,E2 -1905.433} C_VEL
LIN {X 0,Y 581.2,Z 525.809,A -85,B 0,C 180,E1 -1906.103,E2 -1906.103} C_VEL
LIN {X 0,Y 581.358,Z 511.318,A -85,B 0,C 180,E1 -1906.639,E2 -1906.639} C_VEL
LIN {X 0,Y 581.488,Z 496.062,A -85,B 0,C 180,E1 -1907.052,E2 -1907.052} C_VEL
LIN {X 0,Y 581.551,Z 480.545,A -85,B 0,C 180,E1 -1907.323,E2 -1907.323} C_VEL
LIN {X 0,Y 581.801,Z 326.672,A -85,B 0,C 180,E1 -1909.275,E2 -1909.275} C_VEL
LIN {X 0,Y 580.898,Z 321.765,A -85,B 0,C 180,E1 -1909.386,E2 -1909.386} C_VEL
LIN {X 0,Y 581.197,Z 296.397,A -85,B 0,C 180,E1 -1912.389,E2 -1912.389} C_VEL
LIN {X 0,Y 581.423,Z 272.988,A -85,B 0,C 180,E1 -1915.219,E2 -1915.219} C_VEL
LIN {X 0,Y 581.223,Z 269.867,A -85,B 0,C 180,E1 -1915.612,E2 -1915.612} C_VEL
LIN {X 0,Y 580.28,Z 265.832,A -85,B 0,C 180,E1 -1916.172,E2 -1916.172} C_VEL
LIN {X 0,Y 580.292,Z 265.822,A -85,B 0,C 180,E1 -1919.308,E2 -1919.308} C_VEL
LIN {X 0,Y 580.289,Z 265.829,A -85,B 0,C 180,E1 -1922.2,E2 -1922.2} C_VEL
LIN {X 0,Y 580.273,Z 265.825,A -85,B 0,C 180,E1 -1924.696,E2 -1924.696} C_VEL
LIN {X 0,Y 580.268,Z 265.824,A -85,B 0,C 180,E1 -1927.269,E2 -1927.269} C_VEL
LIN {X 0,Y 580.278,Z 265.829,A -85,B 0,C 180,E1 -1930.269,E2 -1930.269} C_VEL
LIN {X 0,Y 580.244,Z 265.828,A -85,B 0,C 180,E1 -1932.708,E2 -1932.708} C_VEL
LIN {X 0,Y 580.241,Z 265.831,A -85,B 0,C 180,E1 -1935.61,E2 -1935.61} C_VEL
LIN {X 0,Y 580.248,Z 265.832,A -85,B 0,C 180,E1 -1938.228,E2 -1938.228} C_VEL
LIN {X 0,Y 580.253,Z 265.826,A -85,B 0,C 180,E1 -1940.963,E2 -1940.963} C_VEL
LIN {X 0,Y 580.227,Z 265.834,A -85,B 0,C 180,E1 -1943.593,E2 -1943.593} C_VEL
LIN {X 0,Y 580.265,Z 265.829,A -85,B 0,C 180,E1 -1946.142,E2 -1946.142} C_VEL
LIN {X 0,Y 580.255,Z 265.825,A -85,B 0,C 180,E1 -1948.613,E2 -1948.613} C_VEL
LIN {X 0,Y 580.272,Z 265.824,A -85,B 0,C 180,E1 -1951.023,E2 -1951.023} C_VEL
LIN {X 0,Y 580.229,Z 265.832,A -85,B 0,C 180,E1 -1954.148,E2 -1954.148} C_VEL
LIN {X 0,Y 580.247,Z 265.827,A -85,B 0,C 180,E1 -1956.441,E2 -1956.441} C_VEL
LIN {X 0,Y 580.253,Z 265.832,A -85,B 0,C 180,E1 -1959.436,E2 -1959.436} C_VEL
LIN {X 0,Y 580.227,Z 265.836,A -85,B 0,C 180,E1 -1961.644,E2 -1961.644} C_VEL
LIN {X 0,Y 580.261,Z 265.825,A -85,B 0,C 180,E1 -1964.546,E2 -1964.546} C_VEL
LIN {X 0,Y 580.271,Z 265.83,A -85,B 0,C 180,E1 -1967.408,E2 -1967.408} C_VEL
LIN {X 0,Y 580.214,Z 265.83,A -85,B 0,C 180,E1 -1970.237,E2 -1970.237} C_VEL
LIN {X 0,Y 580.307,Z 265.822,A -85,B 0,C 180,E1 -1973.044,E2 -1973.044} C_VEL
LIN {X 0,Y 580.232,Z 265.832,A -85,B 0,C 180,E1 -1975.832,E2 -1975.832} C_VEL
LIN {X 0,Y 580.303,Z 265.821,A -85,B 0,C 180,E1 -1977.918,E2 -1977.918} C_VEL
LIN {X 0,Y 580.315,Z 265.819,A -85,B 0,C 180,E1 -1980,E2 -1980} C_VEL
LIN {X 0,Y 580.303,Z 265.82,A -85,B 0,C 180,E1 -1982.777,E2 -1982.777} C_VEL
LIN {X 0,Y 580.306,Z 265.824,A -85,B 0,C 180,E1 -1985.56,E2 -1985.56} C_VEL
LIN {X 0,Y 580.277,Z 265.822,A -85,B 0,C 180,E1 -1988.357,E2 -1988.357} C_VEL
LIN {X 0,Y 580.286,Z 265.831,A -85,B 0,C 180,E1 -1991.191,E2 -1991.191} C_VEL
LIN {X 0,Y 580.275,Z 265.823,A -85,B 0,C 180,E1 -1994.018,E2 -1994.018} C_VEL
LIN {X 0,Y 580.276,Z 265.829,A -85,B 0,C 180,E1 -1996.907,E2 -1996.907} C_VEL
LIN {X 0,Y 580.266,Z 265.822,A -85,B 0,C 180,E1 -1999.824,E2 -1999.824} C_VEL
LIN {X 0,Y 580.271,Z 265.829,A -85,B 0,C 180,E1 -2001.295,E2 -2001.295} C_VEL
LIN {X 0,Y 579.56,Z 265.914,A -85,B 0,C 180,E1 -2001.874,E2 -2001.874} C_VEL
LIN {X 0,Y 576.677,Z 266.275,A -85,B 0,C 180,E1 -2002.814,E2 -2002.814} C_VEL
LIN {X 0,Y 574.28,Z 266.572,A -85,B 0,C 180,E1 -2003.57,E2 -2003.57} C_VEL
LIN {X 0,Y 573.272,Z 266.696,A -85,B 0,C 180,E1 -2004.154,E2 -2004.154} C_VEL
LIN {X 0,Y 573.2,Z 266.705,A -85,B 0,C 180,E1 -2004.352,E2 -2004.352} C_VEL
LIN {X 0,Y 573.238,Z 266.706,A -85,B 0,C 180,E1 -2006.977,E2 -2006.977} C_VEL
LIN {X 0,Y 573.226,Z 266.703,A -85,B 0,C 180,E1 -2009.487,E2 -2009.487} C_VEL
LIN {X 0,Y 573.241,Z 266.704,A -85,B 0,C 180,E1 -2012.646,E2 -2012.646} C_VEL
LIN {X 0,Y 573.2,Z 266.71,A -85,B 0,C 180,E1 -2015.189,E2 -2015.189} C_VEL
LIN {X 0,Y 573.223,Z 266.701,A -85,B 0,C 180,E1 -2017.809,E2 -2017.809} C_VEL
LIN {X 0,Y 573.236,Z 266.704,A -85,B 0,C 180,E1 -2020.526,E2 -2020.526} C_VEL
LIN {X 0,Y 573.229,Z 266.703,A -85,B 0,C 180,E1 -2023.36,E2 -2023.36} C_VEL
LIN {X 0,Y 573.23,Z 266.709,A -85,B 0,C 180,E1 -2026.642,E2 -2026.642} C_VEL
LIN {X 0,Y 573.239,Z 266.7,A -85,B 0,C 180,E1 -2029.476,E2 -2029.476} C_VEL
LIN {X 0,Y 573.227,Z 266.703,A -85,B 0,C 180,E1 -2032.193,E2 -2032.193} C_VEL
LIN {X 0,Y 573.236,Z 266.702,A -85,B 0,C 180,E1 -2035.229,E2 -2035.229} C_VEL
LIN {X 0,Y 573.242,Z 266.703,A -85,B 0,C 180,E1 -2038.186,E2 -2038.186} C_VEL
LIN {X 0,Y 573.256,Z 266.706,A -85,B 0,C 180,E1 -2040.635,E2 -2040.635} C_VEL
LIN {X 0,Y 573.248,Z 266.702,A -85,B 0,C 180,E1 -2043.025,E2 -2043.025} C_VEL
LIN {X 0,Y 573.273,Z 266.699,A -85,B 0,C 180,E1 -2045.367,E2 -2045.367} C_VEL
LIN {X 0,Y 573.283,Z 266.845,A -85,B 0,C 180,E1 -2046.775,E2 -2046.775} C_VEL
LIN {X 0,Y 574.068,Z 271.802,A -85,B 0,C 180,E1 -2047.507,E2 -2047.507} C_VEL
LIN {X 0,Y 573.842,Z 291.773,A -85,B 0,C 180,E1 -2050.281,E2 -2050.281} C_VEL
LIN {X 0,Y 573.855,Z 292.922,A -85,B 0,C 180,E1 -2050.44,E2 -2050.44} C_VEL
LIN {X 0,Y 575.154,Z 299.455,A -85,B 0,C 180,E1 -2050.574,E2 -2050.574} C_VEL
LIN {X 0,Y 574.748,Z 458.073,A -85,B 0,C 180,E1 -2052.625,E2 -2052.625} C_VEL
LIN {X 0,Y 574.604,Z 473.763,A -85,B 0,C 180,E1 -2052.976,E2 -2052.976} C_VEL
LIN {X 0,Y 574.407,Z 489.076,A -85,B 0,C 180,E1 -2053.473,E2 -2053.473} C_VEL
LIN {X 0,Y 574.252,Z 503.734,A -85,B 0,C 180,E1 -2054.108,E2 -2054.108} C_VEL
LIN {X 0,Y 574.03,Z 517.042,A -85,B 0,C 180,E1 -2054.83,E2 -2054.83} C_VEL
LIN {X 0,Y 573.858,Z 530.56,A -85,B 0,C 180,E1 -2055.729,E2 -2055.729} C_VEL
LIN {X 0,Y 573.631,Z 542.886,A -85,B 0,C 180,E1 -2056.72,E2 -2056.72} C_VEL
LIN {X 0,Y 573.462,Z 554.083,A -85,B 0,C 180,E1 -2057.796,E2 -2057.796} C_VEL
LIN {X 0,Y 573.294,Z 563.584,A -85,B 0,C 180,E1 -2058.877,E2 -2058.877} C_VEL
LIN {X 0,Y 573.203,Z 572.778,A -85,B 0,C 180,E1 -2060.116,E2 -2060.116} C_VEL
LIN {X 0,Y 573.134,Z 580.487,A -85,B 0,C 180,E1 -2061.361,E2 -2061.361} C_VEL
LIN {X 0,Y 573.075,Z 586.883,A -85,B 0,C 180,E1 -2062.602,E2 -2062.602} C_VEL
LIN {X 0,Y 573.041,Z 592.767,A -85,B 0,C 180,E1 -2064.016,E2 -2064.016} C_VEL
LIN {X 0,Y 572.95,Z 596.251,A -85,B 0,C 180,E1 -2065.074,E2 -2065.074} C_VEL
LIN {X 0,Y 573.004,Z 599.795,A -85,B 0,C 180,E1 -2066.484,E2 -2066.484} C_VEL
LIN {X 0,Y 572.938,Z 602.139,A -85,B 0,C 180,E1 -2067.891,E2 -2067.891} C_VEL
LIN {X 0,Y 572.936,Z 603.337,A -85,B 0,C 180,E1 -2069.297,E2 -2069.297} C_VEL
LIN {X 0,Y 572.937,Z 603.359,A -85,B 0,C 180,E1 -2070.703,E2 -2070.703} C_VEL
LIN {X 0,Y 572.938,Z 602.243,A -85,B 0,C 180,E1 -2072.109,E2 -2072.109} C_VEL
LIN {X 0,Y 573.006,Z 599.981,A -85,B 0,C 180,E1 -2073.516,E2 -2073.516} C_VEL
LIN {X 0,Y 572.95,Z 596.521,A -85,B 0,C 180,E1 -2074.926,E2 -2074.926} C_VEL
LIN {X 0,Y 573.007,Z 591.788,A -85,B 0,C 180,E1 -2076.337,E2 -2076.337} C_VEL
LIN {X 0,Y 573.094,Z 585.655,A -85,B 0,C 180,E1 -2077.752,E2 -2077.752} C_VEL
LIN {X 0,Y 573.134,Z 577.935,A -85,B 0,C 180,E1 -2079.172,E2 -2079.172} C_VEL
LIN {X 0,Y 573.265,Z 569.696,A -85,B 0,C 180,E1 -2080.418,E2 -2080.418} C_VEL
LIN {X 0,Y 573.358,Z 559.787,A -85,B 0,C 180,E1 -2081.668,E2 -2081.668} C_VEL
LIN {X 0,Y 573.534,Z 549.637,A -85,B 0,C 180,E1 -2082.742,E2 -2082.742} C_VEL
LIN {X 0,Y 573.721,Z 537.559,A -85,B 0,C 180,E1 -2083.82,E2 -2083.82} C_VEL
LIN {X 0,Y 573.918,Z 524.605,A -85,B 0,C 180,E1 -2084.779,E2 -2084.779} C_VEL
LIN {X 0,Y 574.145,Z 510.724,A -85,B 0,C 180,E1 -2085.622,E2 -2085.622} C_VEL
LIN {X 0,Y 574.35,Z 495.794,A -85,B 0,C 180,E1 -2086.346,E2 -2086.346} C_VEL
LIN {X 0,Y 574.552,Z 481.284,A -85,B 0,C 180,E1 -2086.888,E2 -2086.888} C_VEL
LIN {X 0,Y 574.7,Z 465.857,A -85,B 0,C 180,E1 -2087.309,E2 -2087.309} C_VEL
LIN {X 0,Y 574.784,Z 450.79,A -85,B 0,C 180,E1 -2087.575,E2 -2087.575} C_VEL
LIN {X 0,Y 575.096,Z 299.127,A -85,B 0,C 180,E1 -2089.522,E2 -2089.522} C_VEL
LIN {X 0,Y 573.831,Z 292.881,A -85,B 0,C 180,E1 -2089.656,E2 -2089.656} C_VEL
LIN {X 0,Y 574.091,Z 273.792,A -85,B 0,C 180,E1 -2092.302,E2 -2092.302} C_VEL
LIN {X 0,Y 573.851,Z 269.741,A -85,B 0,C 180,E1 -2092.882,E2 -2092.882} C_VEL
LIN {X 0,Y 573.238,Z 266.709,A -85,B 0,C 180,E1 -2093.349,E2 -2093.349} C_VEL
LIN {X 0,Y 573.262,Z 266.699,A -85,B 0,C 180,E1 -2096.189,E2 -2096.189} C_VEL
LIN {X 0,Y 573.233,Z 266.701,A -85,B 0,C 180,E1 -2098.564,E2 -2098.564} C_VEL
LIN {X 0,Y 573.227,Z 266.705,A -85,B 0,C 180,E1 -2100.992,E2 -2100.992} C_VEL
LIN {X 0,Y 573.259,Z 266.707,A -85,B 0,C 180,E1 -2103.523,E2 -2103.523} C_VEL
LIN {X 0,Y 573.237,Z 266.702,A -85,B 0,C 180,E1 -2106.049,E2 -2106.049} C_VEL
LIN {X 0,Y 573.239,Z 266.701,A -85,B 0,C 180,E1 -2108.701,E2 -2108.701} C_VEL
LIN {X 0,Y 573.223,Z 266.708,A -85,B 0,C 180,E1 -2111.592,E2 -2111.592} C_VEL
LIN {X 0,Y 573.215,Z 266.703,A -85,B 0,C 180,E1 -2114.334,E2 -2114.334} C_VEL
LIN {X 0,Y 573.233,Z 266.706,A -85,B 0,C 180,E1 -2117.358,E2 -2117.358} C_VEL
LIN {X 0,Y 573.23,Z 266.701,A -85,B 0,C 180,E1 -2120.391,E2 -2120.391} C_VEL
LIN {X 0,Y 573.243,Z 266.706,A -85,B 0,C 180,E1 -2123.077,E2 -2123.077} C_VEL
LIN {X 0,Y 573.255,Z 266.7,A -85,B 0,C 180,E1 -2125.67,E2 -2125.67} C_VEL
LIN {X 0,Y 573.234,Z 266.699,A -85,B 0,C 180,E1 -2128.184,E2 -2128.184} C_VEL
LIN {X 0,Y 573.246,Z 266.699,A -85,B 0,C 180,E1 -2130.633,E2 -2130.633} C_VEL
LIN {X 0,Y 573.239,Z 266.709,A -85,B 0,C 180,E1 -2133.023,E2 -2133.023} C_VEL
LIN {X 0,Y 573.222,Z 266.706,A -85,B 0,C 180,E1 -2135.364,E2 -2135.364} C_VEL
LIN {X 0,Y 573.211,Z 266.703,A -85,B 0,C 180,E1 -2137.661,E2 -2137.661} C_VEL
LIN {X 0,Y 573.253,Z 266.703,A -85,B 0,C 180,E1 -2140.669,E2 -2140.669} C_VEL
LIN {X 0,Y 573.227,Z 266.701,A -85,B 0,C 180,E1 -2143.621,E2 -2143.621} C_VEL
LIN {X 0,Y 573.209,Z 266.707,A -85,B 0,C 180,E1 -2146.529,E2 -2146.529} C_VEL
LIN {X 0,Y 573.248,Z 266.707,A -85,B 0,C 180,E1 -2148.745,E2 -2148.745} C_VEL
LIN {X 0,Y 573.224,Z 266.701,A -85,B 0,C 180,E1 -2151.54,E2 -2151.54} C_VEL
LIN {X 0,Y 573.197,Z 266.704,A -85,B 0,C 180,E1 -2153.664,E2 -2153.664} C_VEL
LIN {X 0,Y 573.184,Z 266.705,A -85,B 0,C 180,E1 -2155.781,E2 -2155.781} C_VEL
LIN {X 0,Y 573.275,Z 266.695,A -85,B 0,C 180,E1 -2157.892,E2 -2157.892} C_VEL
LIN {X 0,Y 573.322,Z 266.698,A -85,B 0,C 180,E1 -2160.702,E2 -2160.702} C_VEL
LIN {X 0,Y 573.286,Z 266.7,A -85,B 0,C 180,E1 -2162.811,E2 -2162.811} C_VEL
LIN {X 0,Y 573.247,Z 266.698,A -85,B 0,C 180,E1 -2165.629,E2 -2165.629} C_VEL
LIN {X 0,Y 573.198,Z 266.705,A -85,B 0,C 180,E1 -2167.751,E2 -2167.751} C_VEL
LIN {X 0,Y 573.227,Z 266.71,A -85,B 0,C 180,E1 -2170.597,E2 -2170.597} C_VEL
LIN {X 0,Y 573.196,Z 266.704,A -85,B 0,C 180,E1 -2173.471,E2 -2173.471} C_VEL
LIN {X 0,Y 573.202,Z 266.705,A -85,B 0,C 180,E1 -2175.649,E2 -2175.649} C_VEL
LIN {X 0,Y 573.186,Z 266.713,A -85,B 0,C 180,E1 -2178.59,E2 -2178.59} C_VEL
LIN {X 0,Y 573.237,Z 266.699,A -85,B 0,C 180,E1 -2181.291,E2 -2181.291} C_VEL
LIN {X 0,Y 573.198,Z 266.708,A -85,B 0,C 180,E1 -2183.867,E2 -2183.867} C_VEL
LIN {X 0,Y 573.185,Z 266.713,A -85,B 0,C 180,E1 -2186.485,E2 -2186.485} C_VEL
LIN {X 0,Y 573.225,Z 266.701,A -85,B 0,C 180,E1 -2189.368,E2 -2189.368} C_VEL
LIN {X 0,Y 573.236,Z 266.709,A -85,B 0,C 180,E1 -2192.228,E2 -2192.228} C_VEL
LIN {X 0,Y 573.206,Z 266.705,A -85,B 0,C 180,E1 -2194.769,E2 -2194.769} C_VEL
LIN {X 0,Y 573.207,Z 266.708,A -85,B 0,C 180,E1 -2197.81,E2 -2197.81} C_VEL
LIN {X 0,Y 573.235,Z 266.701,A -85,B 0,C 180,E1 -2200.526,E2 -2200.526} C_VEL
LIN {X 0,Y 573.197,Z 266.706,A -85,B 0,C 180,E1 -2203.363,E2 -2203.363} C_VEL
LIN {X 0,Y 573.196,Z 266.71,A -85,B 0,C 180,E1 -2206.336,E2 -2206.336} C_VEL
LIN {X 0,Y 573.197,Z 266.707,A -85,B 0,C 180,E1 -2208.541,E2 -2208.541} C_VEL
LIN {X 0,Y 573.226,Z 266.702,A -85,B 0,C 180,E1 -2211.298,E2 -2211.298} C_VEL
LIN {X 0,Y 573.183,Z 266.715,A -85,B 0,C 180,E1 -2214.022,E2 -2214.022} C_VEL
LIN {X 0,Y 573.247,Z 266.701,A -85,B 0,C 180,E1 -2216.517,E2 -2216.517} C_VEL
LIN {X 0,Y 573.221,Z 266.703,A -85,B 0,C 180,E1 -2219.119,E2 -2219.119} C_VEL
LIN {X 0,Y 573.219,Z 266.708,A -85,B 0,C 180,E1 -2221.435,E2 -2221.435} C_VEL
LIN {X 0,Y 573.224,Z 266.765,A -85,B 0,C 180,E1 -2223.643,E2 -2223.643} C_VEL
LIN {X 0,Y 574.576,Z 272.877,A -85,B 0,C 180,E1 -2224.459,E2 -2224.459} C_VEL
LIN {X 0,Y 574.387,Z 291.326,A -85,B 0,C 180,E1 -2226.712,E2 -2226.712} C_VEL
LIN {X 0,Y 574.085,Z 313.564,A -85,B 0,C 180,E1 -2229.393,E2 -2229.393} C_VEL
LIN {X 0,Y 574.013,Z 321.875,A -85,B 0,C 180,E1 -2230.385,E2 -2230.385} C_VEL
LIN {X 0,Y 575.214,Z 328.48,A -85,B 0,C 180,E1 -2230.518,E2 -2230.518} C_VEL
LIN {X 0,Y 574.753,Z 488.214,A -85,B 0,C 180,E1 -2232.583,E2 -2232.583} C_VEL
LIN {X 0,Y 574.617,Z 503.723,A -85,B 0,C 180,E1 -2232.931,E2 -2232.931} C_VEL
LIN {X 0,Y 574.411,Z 519.052,A -85,B 0,C 180,E1 -2233.428,E2 -2233.428} C_VEL
LIN {X 0,Y 574.292,Z 532.781,A -85,B 0,C 180,E1 -2234.018,E2 -2234.018} C_VEL
LIN {X 0,Y 574.048,Z 546.252,A -85,B 0,C 180,E1 -2234.739,E2 -2234.739} C_VEL
LIN {X 0,Y 573.86,Z 559.824,A -85,B 0,C 180,E1 -2235.632,E2 -2235.632} C_VEL
